REGION Network 16: Timeout
   Label( End_G7 )
   RUNG wire#powerrail
      Contact( #Switching_left )
      wire#w1
      { S7_Templates := "time_type := Time" } #MABS_sw_timout.TON(pt := T#10s, et =>)
      wire#w2
      I_Contact( #MABS.Reset_error )
      I_Contact( #MABS.EMS )
      Coil( #MABS.Error_timeout_sw )
   END_RUNG
   RUNG wire#powerrail
      Contact( #"Switching_left to straight" )
   END_RUNG wire#w1
   RUNG wire#powerrail
      Contact( #"Switching_right to straight" )
   END_RUNG wire#w1
   RUNG wire#powerrail
      Contact( #Switching_right )
   END_RUNG wire#w1
   RUNG wire#powerrail
      Contact( #MABS.Error_timeout_sw )
   END_RUNG wire#w2
   // the same network as SCL:
   End_G7:
   #MABS_sw_timout(IN := #Switching_left OR #"Switching_left to straight" OR #"Switching_right to straight" OR #Switching_right,   // TON
                   PT := T#10s);
   #MABS.Error_timeout_sw := (#MABS_sw_timout.Q OR #MABS.Error_timeout_sw) AND NOT #MABS.Reset_error AND NOT #MABS.EMS;
END_REGION

REGION Network 17: Postion reached + origin sensor
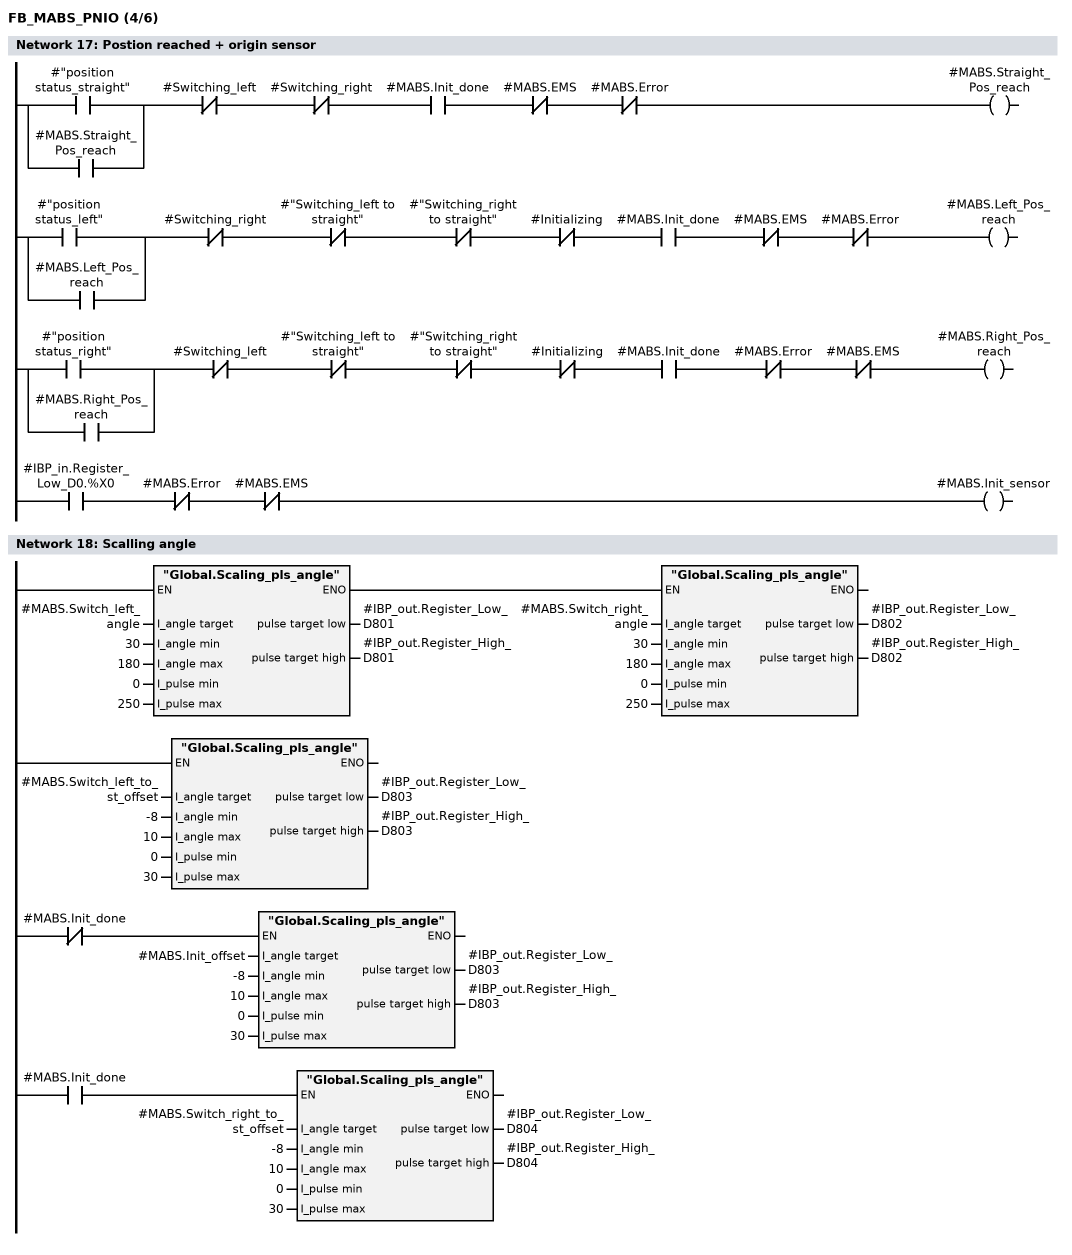
   RUNG wire#powerrail
      Contact( #"position status_straight" )
      wire#w1
      I_Contact( #Switching_left )
      I_Contact( #Switching_right )
      Contact( #MABS.Init_done )
      I_Contact( #MABS.EMS )
      I_Contact( #MABS.Error )
      Coil( #MABS.Straight_Pos_reach )
   END_RUNG
   RUNG wire#powerrail
      Contact( #MABS.Straight_Pos_reach )
   END_RUNG wire#w1
   RUNG wire#powerrail
      Contact( #"position status_left" )
      wire#w2
      I_Contact( #Switching_right )
      I_Contact( #"Switching_left to straight" )
      I_Contact( #"Switching_right to straight" )
      I_Contact( #Initializing )
      Contact( #MABS.Init_done )
      I_Contact( #MABS.EMS )
      I_Contact( #MABS.Error )
      Coil( #MABS.Left_Pos_reach )
   END_RUNG
   RUNG wire#powerrail
      Contact( #MABS.Left_Pos_reach )
   END_RUNG wire#w2
   RUNG wire#powerrail
      Contact( #"position status_right" )
      wire#w3
      I_Contact( #Switching_left )
      I_Contact( #"Switching_left to straight" )
      I_Contact( #"Switching_right to straight" )
      I_Contact( #Initializing )
      Contact( #MABS.Init_done )
      I_Contact( #MABS.Error )
      I_Contact( #MABS.EMS )
      Coil( #MABS.Right_Pos_reach )
   END_RUNG
   RUNG wire#powerrail
      Contact( #MABS.Right_Pos_reach )
   END_RUNG wire#w3
   RUNG wire#powerrail
      Contact( #IBP_in.Register_Low_D0.%X0 )
      I_Contact( #MABS.Error )
      I_Contact( #MABS.EMS )
      Coil( #MABS.Init_sensor )
   END_RUNG
   // the same network as SCL:
   #MABS.Straight_Pos_reach := (#"position status_straight" OR #MABS.Straight_Pos_reach) AND NOT #Switching_left AND NOT #Switching_right AND #MABS.Init_done AND NOT #MABS.EMS AND NOT #MABS.Error;
   #MABS.Left_Pos_reach := (#"position status_left" OR #MABS.Left_Pos_reach) AND NOT #Switching_right AND NOT #"Switching_left to straight" AND NOT #"Switching_right to straight" AND NOT #Initializing AND #MABS.Init_done AND NOT #MABS.EMS AND NOT #MABS.Error;
   #MABS.Right_Pos_reach := (#"position status_right" OR #MABS.Right_Pos_reach) AND NOT #Switching_left AND NOT #"Switching_left to straight" AND NOT #"Switching_right to straight" AND NOT #Initializing AND #MABS.Init_done AND NOT #MABS.Error AND NOT #MABS.EMS;
   #MABS.Init_sensor := #IBP_in.Register_Low_D0.%X0 AND NOT #MABS.Error AND NOT #MABS.EMS;
END_REGION

REGION Network 18: Scalling angle
   RUNG wire#powerrail
      "Global.Scaling_pls_angle"("I_angle target" := #MABS.Switch_left_angle, "I_angle min" := 30, "I_angle max" := 180, "I_pulse min" := 0, "I_pulse max" := 250, "pulse target low" => #IBP_out.Register_Low_D801, "pulse target high" => #IBP_out.Register_High_D801)
      "Global.Scaling_pls_angle"("I_angle target" := #MABS.Switch_right_angle, "I_angle min" := 30, "I_angle max" := 180, "I_pulse min" := 0, "I_pulse max" := 250, "pulse target low" => #IBP_out.Register_Low_D802, "pulse target high" => #IBP_out.Register_High_D802)
   END_RUNG
   RUNG wire#powerrail
      "Global.Scaling_pls_angle"("I_angle target" := #MABS.Switch_left_to_st_offset, "I_angle min" := -8, "I_angle max" := 10, "I_pulse min" := 0, "I_pulse max" := 30, "pulse target low" => #IBP_out.Register_Low_D803, "pulse target high" => #IBP_out.Register_High_D803)
   END_RUNG
   RUNG wire#powerrail
      I_Contact( #MABS.Init_done )
      "Global.Scaling_pls_angle"("I_angle target" := #MABS.Init_offset, "I_angle min" := -8, "I_angle max" := 10, "I_pulse min" := 0, "I_pulse max" := 30, "pulse target low" => #IBP_out.Register_Low_D803, "pulse target high" => #IBP_out.Register_High_D803)
   END_RUNG
   RUNG wire#powerrail
      Contact( #MABS.Init_done )
      "Global.Scaling_pls_angle"("I_angle target" := #MABS.Switch_right_to_st_offset, "I_angle min" := -8, "I_angle max" := 10, "I_pulse min" := 0, "I_pulse max" := 30, "pulse target low" => #IBP_out.Register_Low_D804, "pulse target high" => #IBP_out.Register_High_D804)
   END_RUNG
   // the same network as SCL:
   "Global.Scaling_pls_angle"("I_angle target" := #MABS.Switch_left_angle,
                           "I_angle min" := 30,
                           "I_angle max" := 180,
                           "I_pulse min" := 0,
                           "I_pulse max" := 250,
                           "pulse target low" => #IBP_out.Register_Low_D801,
                           "pulse target high" => #IBP_out.Register_High_D801,
                           ENO => #_w1);
   IF #_w1 THEN
       "Global.Scaling_pls_angle"("I_angle target" := #MABS.Switch_right_angle,
                               "I_angle min" := 30,
                               "I_angle max" := 180,
                               "I_pulse min" := 0,
                               "I_pulse max" := 250,
                               "pulse target low" => #IBP_out.Register_Low_D802,
                               "pulse target high" => #IBP_out.Register_High_D802);
   END_IF;
   "Global.Scaling_pls_angle"("I_angle target" := #MABS.Switch_left_to_st_offset,
                           "I_angle min" := -8,
                           "I_angle max" := 10,
                           "I_pulse min" := 0,
                           "I_pulse max" := 30,
                           "pulse target low" => #IBP_out.Register_Low_D803,
                           "pulse target high" => #IBP_out.Register_High_D803);
   IF NOT #MABS.Init_done THEN
       "Global.Scaling_pls_angle"("I_angle target" := #MABS.Init_offset,
                               "I_angle min" := -8,
                               "I_angle max" := 10,
                               "I_pulse min" := 0,
                               "I_pulse max" := 30,
                               "pulse target low" => #IBP_out.Register_Low_D803,
                               "pulse target high" => #IBP_out.Register_High_D803);
   END_IF;
   IF #MABS.Init_done THEN
       "Global.Scaling_pls_angle"("I_angle target" := #MABS.Switch_right_to_st_offset,
                               "I_angle min" := -8,
                               "I_angle max" := 10,
                               "I_pulse min" := 0,
                               "I_pulse max" := 30,
                               "pulse target low" => #IBP_out.Register_Low_D804,
                               "pulse target high" => #IBP_out.Register_High_D804);
   END_IF;
END_REGION

REGION Network 19: Swing direction
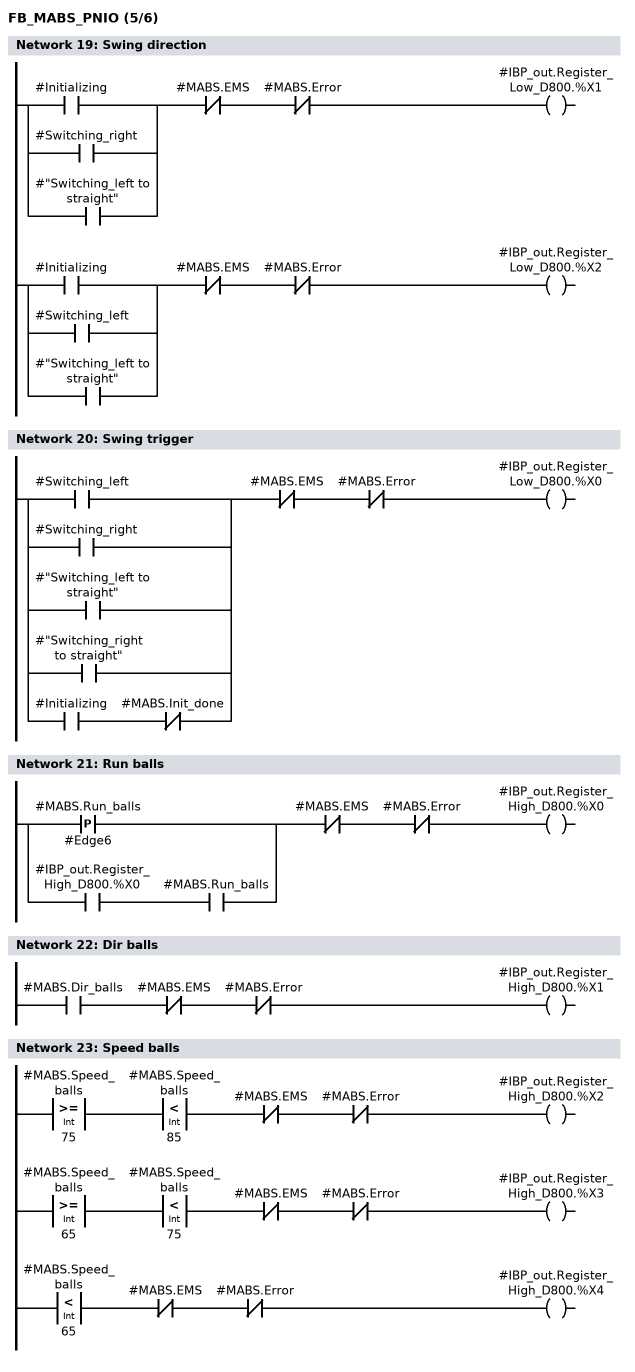
   RUNG wire#powerrail
      Contact( #Initializing )
      wire#w1
      I_Contact( #MABS.EMS )
      I_Contact( #MABS.Error )
      Coil( #IBP_out.Register_Low_D800.%X1 )
   END_RUNG
   RUNG wire#powerrail
      Contact( #Switching_right )
   END_RUNG wire#w1
   RUNG wire#powerrail
      Contact( #"Switching_left to straight" )
   END_RUNG wire#w1
   RUNG wire#powerrail
      Contact( #Initializing )
      wire#w2
      I_Contact( #MABS.EMS )
      I_Contact( #MABS.Error )
      Coil( #IBP_out.Register_Low_D800.%X2 )
   END_RUNG
   RUNG wire#powerrail
      Contact( #Switching_left )
   END_RUNG wire#w2
   RUNG wire#powerrail
      Contact( #"Switching_left to straight" )
   END_RUNG wire#w2
   // the same network as SCL:
   #IBP_out.Register_Low_D800.%X1 := (#Initializing OR #Switching_right OR #"Switching_left to straight") AND NOT #MABS.EMS AND NOT #MABS.Error;
   #IBP_out.Register_Low_D800.%X2 := (#Initializing OR #Switching_left OR #"Switching_left to straight") AND NOT #MABS.EMS AND NOT #MABS.Error;
END_REGION

REGION Network 20: Swing trigger
   RUNG wire#powerrail
      Contact( #Switching_left )
      wire#w1
      I_Contact( #MABS.EMS )
      I_Contact( #MABS.Error )
      Coil( #IBP_out.Register_Low_D800.%X0 )
   END_RUNG
   RUNG wire#powerrail
      Contact( #Switching_right )
   END_RUNG wire#w1
   RUNG wire#powerrail
      Contact( #"Switching_left to straight" )
   END_RUNG wire#w1
   RUNG wire#powerrail
      Contact( #"Switching_right to straight" )
   END_RUNG wire#w1
   RUNG wire#powerrail
      Contact( #Initializing )
      I_Contact( #MABS.Init_done )
   END_RUNG wire#w1
   // the same network as SCL:
   #IBP_out.Register_Low_D800.%X0 := (#Switching_left OR #Switching_right OR #"Switching_left to straight" OR #"Switching_right to straight" OR (#Initializing AND NOT #MABS.Init_done)) AND NOT #MABS.EMS AND NOT #MABS.Error;
END_REGION

REGION Network 21: Run balls
   RUNG wire#powerrail
      P_Contact(operand := #MABS.Run_balls, bit := #Edge6)
      wire#w1
      I_Contact( #MABS.EMS )
      I_Contact( #MABS.Error )
      Coil( #IBP_out.Register_High_D800.%X0 )
   END_RUNG
   RUNG wire#powerrail
      Contact( #IBP_out.Register_High_D800.%X0 )
      Contact( #MABS.Run_balls )
   END_RUNG wire#w1
   // the same network as SCL:
   #_w1 := #MABS.Run_balls AND NOT #Edge6;   // rising edge of #MABS.Run_balls
   #Edge6 := #MABS.Run_balls;
   #IBP_out.Register_High_D800.%X0 := (#_w1 OR (#IBP_out.Register_High_D800.%X0 AND #MABS.Run_balls)) AND NOT #MABS.EMS AND NOT #MABS.Error;
END_REGION

REGION Network 22: Dir balls
   RUNG wire#powerrail
      Contact( #MABS.Dir_balls )
      I_Contact( #MABS.EMS )
      I_Contact( #MABS.Error )
      Coil( #IBP_out.Register_High_D800.%X1 )
   END_RUNG
   // the same network as SCL:
   #IBP_out.Register_High_D800.%X1 := #MABS.Dir_balls AND NOT #MABS.EMS AND NOT #MABS.Error;
END_REGION

REGION Network 23: Speed balls
   RUNG wire#powerrail
      { S7_Templates := "SrcType := Int" } GE_Contact(in1 := #MABS.Speed_balls, in2 := 75)
      { S7_Templates := "SrcType := Int" } LT_Contact(in1 := #MABS.Speed_balls, in2 := 85)
      I_Contact( #MABS.EMS )
      I_Contact( #MABS.Error )
      Coil( #IBP_out.Register_High_D800.%X2 )
   END_RUNG
   RUNG wire#powerrail
      { S7_Templates := "SrcType := Int" } GE_Contact(in1 := #MABS.Speed_balls, in2 := 65)
      { S7_Templates := "SrcType := Int" } LT_Contact(in1 := #MABS.Speed_balls, in2 := 75)
      I_Contact( #MABS.EMS )
      I_Contact( #MABS.Error )
      Coil( #IBP_out.Register_High_D800.%X3 )
   END_RUNG
   RUNG wire#powerrail
      { S7_Templates := "SrcType := Int" } LT_Contact(in1 := #MABS.Speed_balls, in2 := 65)
      I_Contact( #MABS.EMS )
      I_Contact( #MABS.Error )
      Coil( #IBP_out.Register_High_D800.%X4 )
   END_RUNG
   // the same network as SCL:
   #IBP_out.Register_High_D800.%X2 := (#MABS.Speed_balls >= 75) AND (#MABS.Speed_balls < 85) AND NOT #MABS.EMS AND NOT #MABS.Error;
   #IBP_out.Register_High_D800.%X3 := (#MABS.Speed_balls >= 65) AND (#MABS.Speed_balls < 75) AND NOT #MABS.EMS AND NOT #MABS.Error;
   #IBP_out.Register_High_D800.%X4 := (#MABS.Speed_balls < 65) AND NOT #MABS.EMS AND NOT #MABS.Error;
END_REGION

REGION Network 24: HMI status
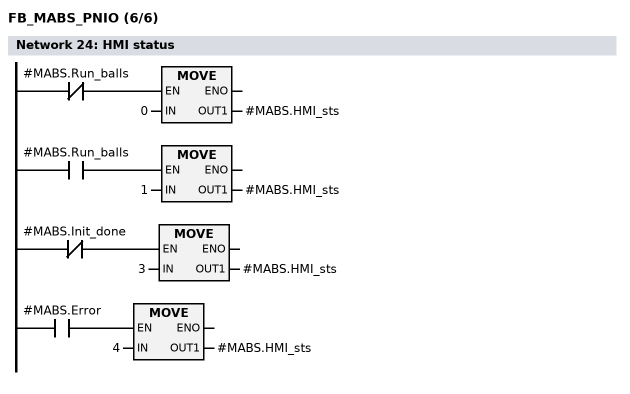
   RUNG wire#powerrail
      I_Contact( #MABS.Run_balls )
      Move(in := 0, out1 => #MABS.HMI_sts)
   END_RUNG
   RUNG wire#powerrail
      Contact( #MABS.Run_balls )
      Move(in := 1, out1 => #MABS.HMI_sts)
   END_RUNG
   RUNG wire#powerrail
      I_Contact( #MABS.Init_done )
      Move(in := 3, out1 => #MABS.HMI_sts)
   END_RUNG
   RUNG wire#powerrail
      Contact( #MABS.Error )
      Move(in := 4, out1 => #MABS.HMI_sts)
   END_RUNG
   // the same network as SCL:
   IF NOT #MABS.Run_balls THEN #MABS.HMI_sts := 0; END_IF;
   IF #MABS.Run_balls THEN #MABS.HMI_sts := 1; END_IF;
   IF NOT #MABS.Init_done THEN #MABS.HMI_sts := 3; END_IF;
   IF #MABS.Error THEN #MABS.HMI_sts := 4; END_IF;
END_REGION
END_FUNCTION_BLOCK

FUNCTION "Scaling_pls_angle" : Void   // FC12, LAD
// stored: Namespace Global, SetENOAutomatically false
   VAR_INPUT
      "I_angle target" : Int;
      "I_angle min" : Int;
      "I_angle max" : Int;
      "I_pulse min" : Int;
      "I_pulse max" : Int;
   END_VAR
   VAR_OUTPUT
      "pulse target low" : Byte;
      "pulse target high" : Byte;
   END_VAR
   VAR_TEMP
      R_pulse_calcul : Real;
      R_angle_calcul : Real;
      pulse_target_int : Int;
      Int4 : Int;
      Int5 : Int;
      Real1 : Real;
      Real2 : Real;
      Real3 : Real;
      Real4 : Real;
   END_VAR
BEGIN

REGION Network 1: Convert diff in real
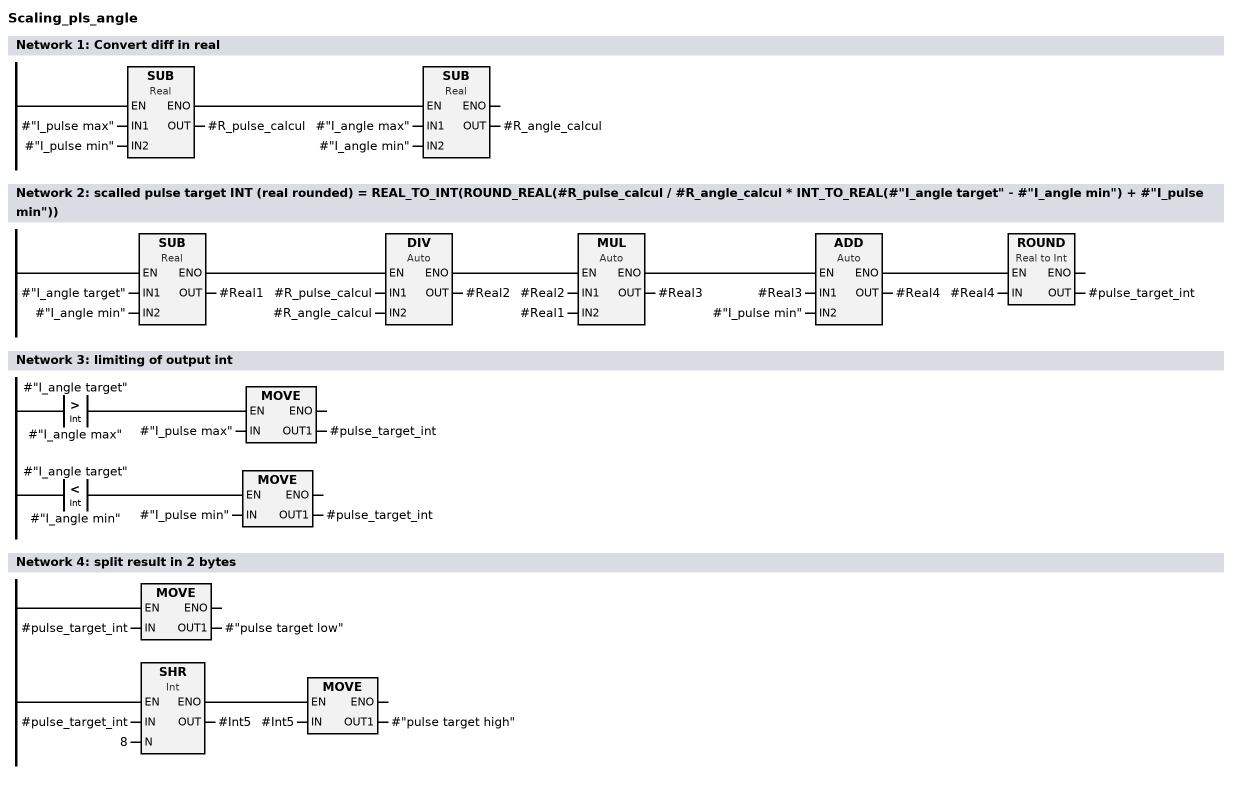
   RUNG wire#powerrail
      { S7_Templates := "SrcType := Real" } Sub(in1 := #"I_pulse max", in2 := #"I_pulse min", out => #R_pulse_calcul)
      { S7_Templates := "SrcType := Real" } Sub(in1 := #"I_angle max", in2 := #"I_angle min", out => #R_angle_calcul)
   END_RUNG
   // the same network as SCL:
   #R_pulse_calcul := #"I_pulse max" - #"I_pulse min";
   #R_angle_calcul := #"I_angle max" - #"I_angle min";
END_REGION

REGION Network 2: scalled pulse target INT (real rounded) = REAL_TO_INT(ROUND_REAL(#R_pulse_calcul / #R_angle_calcul * INT_TO_REAL(#"I_angle target" - #"I_angle min") + #"I_pulse min"))
   RUNG wire#powerrail
      { S7_Templates := "SrcType := Real" } Sub(in1 := #"I_angle target", in2 := #"I_angle min", out => #Real1)
      Div(in1 := #R_pulse_calcul, in2 := #R_angle_calcul, out => #Real2)
      Mul(in1 := #Real2, in2 := #Real1, out => #Real3)
      Add(in1 := #Real3, in2 := #"I_pulse min", out => #Real4)
      { S7_Templates := "[SrcType := Real, DestType := Int]" } Round(in := #Real4, out => #pulse_target_int)
   END_RUNG
   // the same network as SCL:
   #Real1 := #"I_angle target" - #"I_angle min";
   #Real2 := #R_pulse_calcul / #R_angle_calcul;
   #Real3 := #Real2 * #Real1;
   #Real4 := #Real3 + #"I_pulse min";
   #pulse_target_int := ROUND(#Real4);
END_REGION

REGION Network 3: limiting of output int
   RUNG wire#powerrail
      { S7_Templates := "SrcType := Int" } GT_Contact(in1 := #"I_angle target", in2 := #"I_angle max")
      Move(in := #"I_pulse max", out1 => #pulse_target_int)
   END_RUNG
   RUNG wire#powerrail
      { S7_Templates := "SrcType := Int" } LT_Contact(in1 := #"I_angle target", in2 := #"I_angle min")
      Move(in := #"I_pulse min", out1 => #pulse_target_int)
   END_RUNG
   // the same network as SCL:
   IF #"I_angle target" > #"I_angle max" THEN #pulse_target_int := #"I_pulse max"; END_IF;
   IF #"I_angle target" < #"I_angle min" THEN #pulse_target_int := #"I_pulse min"; END_IF;
END_REGION

REGION Network 4: split result in 2 bytes
   RUNG wire#powerrail
      Move(in := #pulse_target_int, out1 => #"pulse target low")
   END_RUNG
   RUNG wire#powerrail
      { S7_Templates := "SrcType := Int" } Shr(in := #pulse_target_int, n := 8, out => #Int5)
      Move(in := #Int5, out1 => #"pulse target high")
   END_RUNG
   // the same network as SCL:
   #"pulse target low" := #pulse_target_int;
   #Int5 := SHR(IN := #pulse_target_int, N := 8);
   #"pulse target high" := #Int5;
END_REGION
END_FUNCTION

FUNCTION_BLOCK "FB_ManualControl"   // FB37, LAD
// stored: Access Published, MemoryReserve 100, Namespace Global, SetENOAutomatically false
   VAR RETAIN
      "Counter" { S7_SetPoint := 'True'} : CTU_INT;
   END_VAR
BEGIN

REGION Network 1
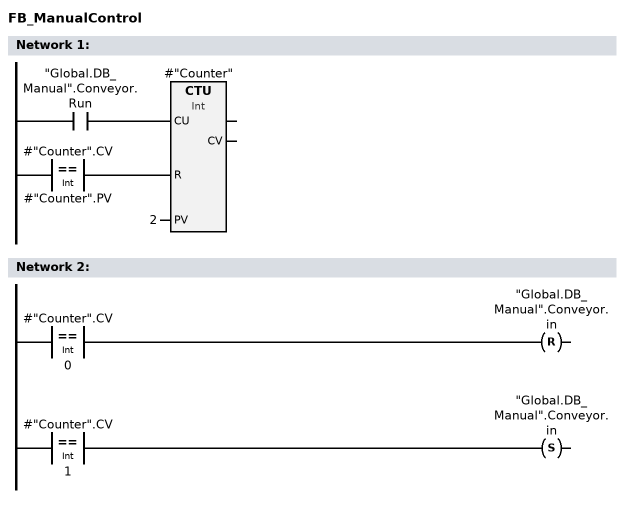
   RUNG wire#powerrail
      Contact( "Global.DB_Manual".Conveyor.Run )
      { S7_Templates := "value_type := Int" } #"Counter".CTU(r := wire#w1, pv := 2, cv =>)
   END_RUNG
   RUNG wire#powerrail
      { S7_Templates := "SrcType := Int" } EQ_Contact(in1 := #"Counter".CV, in2 := #"Counter".PV)
   END_RUNG wire#w1
   // the same network as SCL:
   #"Counter"(CU := "Global.DB_Manual".Conveyor.Run, R := #"Counter".CV = #"Counter".PV, PV := 2);   // CTU
END_REGION

REGION Network 2
   RUNG wire#powerrail
      { S7_Templates := "SrcType := Int" } EQ_Contact(in1 := #"Counter".CV, in2 := 0)
      R_Coil( "Global.DB_Manual".Conveyor.in )
   END_RUNG
   RUNG wire#powerrail
      { S7_Templates := "SrcType := Int" } EQ_Contact(in1 := #"Counter".CV, in2 := 1)
      S_Coil( "Global.DB_Manual".Conveyor.in )
   END_RUNG
   // the same network as SCL:
   IF #"Counter".CV = 0 THEN "Global.DB_Manual".Conveyor.in := FALSE; END_IF;
   IF #"Counter".CV = 1 THEN "Global.DB_Manual".Conveyor.in := TRUE; END_IF;
END_REGION
END_FUNCTION_BLOCK

FUNCTION "FC_SafetyStandard" : Void
{ S7_Optimized_Access := 'TRUE' ; Published := 'TRUE' }
VERSION : 0.1

BEGIN
END_FUNCTION

NAMESPACE Global
ORGANIZATION_BLOCK Main_OB
TITLE = "Main Program Sweep (Cycle)"
{ S7_Optimized_Access := 'TRUE' ; Published := 'FALSE' }
VERSION : 0.1

BEGIN
	// ===
	// GoW
	// ==========================================================================================================================================
	// Company        : LogTech, s.r.o.
	// Created by     : Anton Vinoth Soundraraj
	// Block          : Main_OB
	// Project        : Lékarna DC Chrudim
	// Project number : 23-157
	// ==========================================================================================================================================
	
	REGION System
	    
	    FC_ReadSystemSSR();
	    
	END_REGION
	
	REGION Hardware diag
	    
	    IDB_HardwareDiag();
	    
	END_REGION
	
	REGION Klaxon
	    
	    FC_AllKlaxon();
	    
	END_REGION
	
	REGION Devices
	    
	    IDB_DataMan262(TriggerSignal:=DB_SystemSimu.TriggerSensor.Line.C1.Conveyor[3001],
	                   "Dataman-Results Available":=_."Dataman-Results Available",
	                   "Dataman-TriggerReady":=_."Dataman-TriggerReady",
	                   "Dataman-TriggerAck":=_."Dataman-TriggerAck",
	                   "Dataman-ResultID":=_."Dataman-ResultID",
	                   "Dataman-Result Code":=_."Dataman-Result Code",
	                   "Dataman-Result Length":=_."Dataman-Result Length",
	                   "Result Data":=_."Result Data",
	                   "Dataman-UserData Length"=>_."Dataman-UserData Length",
	                   "Dataman-UserData Option"=>_."Dataman-UserData Option",
	                   "User Data"=>_."User Data",
	                   "Dataman-TriggerEnable":=_."Dataman-TriggerEnable",
	                   "Dataman-Trigger":=_."Dataman-Trigger",
	                   "Dataman-ResultsAck":=_."Dataman-ResultsAck");
	    
	END_REGION
	
END_ORGANIZATION_BLOCK
END_NAMESPACE

NAMESPACE LineA1
FUNCTION_BLOCK FB_LineA1
{ S7_Optimized_Access := 'TRUE' ; Published := 'TRUE' }
VERSION : 0.1
   VAR 
      "Conveyor_A1.1.1" { S7_SetPoint := 'False'} : _.Global.FB_Conveyor;
      "MABS_A1.1.1" { S7_SetPoint := 'False'} : _.Global.FB_MABS;
      "Transfer_A1.1.1" { S7_SetPoint := 'False'} : _.Global.FB_S300_tTransMode;
   END_VAR


BEGIN
	
	
	
	
	
	
	
	
	
	
	
	
	
	
	
END_FUNCTION_BLOCK
END_NAMESPACE

NAMESPACE LineA1
ORGANIZATION_BLOCK Main_LineA1
TITLE = "Main Program Sweep (Cycle)"
{ S7_Optimized_Access := 'TRUE' ; Published := 'FALSE' }
VERSION : 0.1

BEGIN
	IDB_LineA1();
	
END_ORGANIZATION_BLOCK
END_NAMESPACE

NAMESPACE LineB1
FUNCTION_BLOCK FB_LineB1
{ S7_Optimized_Access := 'TRUE' ; Published := 'TRUE' }
VERSION : 0.1
   VAR 
      "Conveyor_B1.1.1" { S7_SetPoint := 'False'} : _.Global.FB_Conveyor;
      "MABS_B1.1.1" { S7_SetPoint := 'False'} : _.Global.FB_MABS;
      "Transfer_B1.1.1" { S7_SetPoint := 'False'} : _.Global.FB_S300_tTransMode;
      "Transfer_B1.1.2" { S7_SetPoint := 'False'} : FB_S300_FullControl;
   END_VAR


BEGIN
	
	
	
	
	
	
	
	
	
	
	
	
	
	
	
END_FUNCTION_BLOCK
END_NAMESPACE

NAMESPACE LineB1
ORGANIZATION_BLOCK Main_LineB1
TITLE = "Main Program Sweep (Cycle)"
{ S7_Optimized_Access := 'TRUE' ; Published := 'FALSE' }
VERSION : 0.1

BEGIN
	IDB_LineB1();
	
END_ORGANIZATION_BLOCK
END_NAMESPACE

NAMESPACE LineC1
FUNCTION_BLOCK FB_LineC1
{ S7_Optimized_Access := 'TRUE' ; Published := 'TRUE' }
VERSION : 0.1
   VAR 
      "Conveyor_C1.1.1" { S7_SetPoint := 'False'} : _.Global.FB_Conveyor;
      "Conveyor_C1.1.2" : _.Global.FB_Conveyor;
      "Conveyor_C1.1.3" : _.Global.FB_Conveyor;
      "MABS_C1.2.1" { S7_SetPoint := 'False'} : _.Global.FB_MABS;
      "MABS_C1.2.2" : _.Global.FB_MABS;
      "Conveyor_C1.3.1" : _.Global.FB_Conveyor;
      "Conveyor_C1.3.2" : _.Global.FB_Conveyor;
      "Conveyor_C1.3.3" : _.Global.FB_Conveyor;
      "Conveyor_C1.3.4" : _.Global.FB_Conveyor;
      "Conveyor_C1.3.5" : _.Global.FB_Conveyor;
      "Conveyor_C1.3.6" : _.Global.FB_Conveyor;
      "Conveyor_C1.3.7" : _.Global.FB_Conveyor;
      "Conveyor_C1.3.8" : _.Global.FB_Conveyor;
      "Conveyor_C1.3.9" : _.Global.FB_Conveyor;
      "Conveyor_C1.3.10" : _.Global.FB_Conveyor;
      "Conveyor_C1.4.1" : _.Global.FB_Conveyor;
      "Conveyor_C1.4.2" : _.Global.FB_Conveyor;
      "Conveyor_C1.4.3" : _.Global.FB_Conveyor;
      "Conveyor_C1.4.4" : _.Global.FB_Conveyor;
      "Conveyor_C1.5.1" : _.Global.FB_Conveyor;
      "Conveyor_C1.6.1" : _.Global.FB_Conveyor;
      "Conveyor_C1.6.2" : _.Global.FB_Conveyor;
      "Conveyor_C1.7.1" : _.Global.FB_Conveyor;
      "Conveyor_C1.7.2" : _.Global.FB_Conveyor;
      "Conveyor_C1.7.3" : _.Global.FB_Conveyor;
      "Conveyor_C1.7.4" : _.Global.FB_Conveyor;
      "Conveyor_C1.7.5" : _.Global.FB_Conveyor;
      "Conveyor_C1.7.6" : _.Global.FB_Conveyor;
      "Conveyor_C1.7.7" : _.Global.FB_Conveyor;
      "Conveyor_C1.7.8" : _.Global.FB_Conveyor;
      "Conveyor_C1.7.9" : _.Global.FB_Conveyor;
      "Conveyor_C1.7.10" : _.Global.FB_Conveyor;
      "Conveyor_C1.8.0" : _.Global.FB_Conveyor;
      "Conveyor_C1.9.1" : _.Global.FB_Conveyor;
      "Conveyor_C1.10.1" : _.Global.FB_Conveyor;
      "Conveyor_C1.11.1" : _.Global.FB_Conveyor;
      "Conveyor_C1.11.2" : _.Global.FB_Conveyor;
      "Conveyor_C1.12.1" : _.Global.FB_Conveyor;
      "Conveyor_C1.12.2" : _.Global.FB_Conveyor;
      "Conveyor_C1.12.3" : _.Global.FB_Conveyor;
      "Transfer_C1.13.1" { S7_SetPoint := 'False'} : _.Global.FB_S300_tTransMode;
      "Transfer_C1.14.1" : _.Global.FB_S300_tTransMode;
      "Conveyor_C1.15.2" : _.Global.FB_Conveyor;
      "Conveyor_C1.15.3" : _.Global.FB_Conveyor;
      "Conveyor_C1.15.4" : _.Global.FB_Conveyor;
      "Conveyor_C1.16.1" : _.Global.FB_Conveyor;
      "Conveyor_C1.17.0" : _.Global.FB_Conveyor;
      "Conveyor_C1.18.1" : _.Global.FB_Conveyor;
      "Conveyor_C1.18.2" : _.Global.FB_Conveyor;
      "Conveyor_C1.18.3" : _.Global.FB_Conveyor;
      "Conveyor_C1.18.4" : _.Global.FB_Conveyor;
      "Conveyor_C1.18.5" : _.Global.FB_Conveyor;
      "Conveyor_C1.18.6" : _.Global.FB_Conveyor;
      "Conveyor_C1.18.7" : _.Global.FB_Conveyor;
      "Conveyor_C1.19.1" : _.Global.FB_Conveyor;
      "Conveyor_C1.20.2" : _.Global.FB_Conveyor;
   END_VAR


BEGIN
	// ==========================================================================================================================================
	// Company        : LogTech, s.r.o.
	// Created by     : Mahmoud Elnady
	// Block          : FC_UpstreaProductionTote
	// Project        : Lekarna, Chrudim -PLC001 -MCC001
	// Project number : 23-157
	// ==========================================================================================================================================
	//start this comment 
	REGION Conveyor_C1.1.1
	    #"Conveyor_C1.1.1"(ConveyorID := _."Conveyor_C1.1.1",
	                       Fault := _.LineC1.DB_UDI.LineC1.Fault.Conveyor[_."Conveyor_C1.1.1"],
	                       Upstream := _.LineC1.DB_UDI.LineC1.Upstream.Conveyor[_."Conveyor_C1.1.1"],
	                       Downstream := _.LineC1.DB_UDI.LineC1.DownstreamAccu.Conveyor[_."Conveyor_C1.1.1"],
	                       Interlock := _.LineC1.DB_UDI.LineC1.Interlock.Conveyor[_."Conveyor_C1.1.1"]);
	END_REGION
	
	
	
	
	REGION Conveyor_C1.1.2
	    #"Conveyor_C1.1.2"(ConveyorID := _."Conveyor_C1.1.2",
	                       Fault := _.LineC1.DB_UDI.LineC1.Fault.Conveyor[_."Conveyor_C1.1.2"],
	                       Upstream := _.LineC1.DB_UDI.LineC1.Upstream.Conveyor[_."Conveyor_C1.1.2"],
	                       Downstream := _.LineC1.DB_UDI.LineC1.DownstreamAccu.Conveyor[_."Conveyor_C1.1.2"],
	                       Interlock := _.LineC1.DB_UDI.LineC1.Interlock.Conveyor[_."Conveyor_C1.1.2"]);
	    ;
	END_REGION
	
	
	
	REGION Conveyor_C1.1.3
	    #"Conveyor_C1.1.3"(ConveyorID := _."Conveyor_C1.1.3",
	                       Fault := _.LineC1.DB_UDI.LineC1.Fault.Conveyor[_."Conveyor_C1.1.3"],
	                       Upstream := _.LineC1.DB_UDI.LineC1.Upstream.Conveyor[_."Conveyor_C1.1.3"],
	                       Downstream := _.LineC1.DB_UDI.LineC1.DownstreamAccu.Conveyor[_."Conveyor_C1.1.3"],
	                       Interlock := _.LineC1.DB_UDI.LineC1.Interlock.Conveyor[_."Conveyor_C1.1.3"]);
	    ;
	END_REGION
	
	
	
	REGION MABS_C1.2.1
	    #"MABS_C1.2.1"(MABS_ID:=_."MABS_C1.2.1",
	                   CrossSensor:=false,
	                   Fault:=_.LineC1.DB_UDI.LineC1.Fault.Conveyor[_."MABS_C1.2.1"],
	                   UpstreamRunning:= #"Conveyor_C1.1.3".ReadConveyorStatus.Running,
	                   Downstream_Straight:=#"Conveyor_C1.3.1".FilteredSensor,
	                   "Downstream_Right/Left":=#"Conveyor_C1.9.1".FilteredSensor,
	                   SortDir:= _.Global.DB_ToteTracking.Conveyor[_."MABS_C1.2.1"].ToteDir,
	                   Setpoints:=DB_ConveyorParameters.Line.C1.MABS[_."MABS_C1.2.1"],
	                   MABS_IBP_in:=_."MABS_C1.2.1_IN",
	                   MABS_IBP_out:=_."MABS_C1.2.1_Out");
	END_REGION
	
	
	
	REGION MABS_C1.2.2
	    #"MABS_C1.2.2"(MABS_ID := _."MABS_C1.2.2",
	                   CrossSensor := false,
	                   Fault := _.LineC1.DB_UDI.LineC1.Fault.Conveyor[_."MABS_C1.2.2"],
	                   UpstreamRunning := #"Conveyor_C1.1.3".ReadConveyorStatus.Running,
	                   Downstream_Straight := #"Conveyor_C1.3.1".FilteredSensor,
	                   "Downstream_Right/Left" := #"Conveyor_C1.9.1".FilteredSensor,
	                   SortDir := _.Global.DB_ToteTracking.Conveyor[_."MABS_C1.2.2"].ToteDir,
	                   Setpoints := DB_ConveyorParameters.Line.C1.MABS[_."MABS_C1.2.2"],
	                   MABS_IBP_in := _."MABS_C1.2.2_IN",
	                   MABS_IBP_out := _."MABS_C1.2.2_Out");
	END_REGION
	
	
	REGION Conveyor_C1.3.1
	    #"Conveyor_C1.3.1"(ConveyorID := _."Conveyor_C1.3.1",
	                       Fault := _.LineC1.DB_UDI.LineC1.Fault.Conveyor[_."Conveyor_C1.3.1"],
	                       Upstream := _.LineC1.DB_UDI.LineC1.Upstream.Conveyor[_."Conveyor_C1.3.1"],
	                       Downstream := _.LineC1.DB_UDI.LineC1.DownstreamAccu.Conveyor[_."Conveyor_C1.3.1"],
	                       Interlock := _.LineC1.DB_UDI.LineC1.Interlock.Conveyor[_."Conveyor_C1.3.1"]);
	    ;
	END_REGION
	
	
	REGION Conveyor_C1.3.2
	    #"Conveyor_C1.3.2"(ConveyorID := _."Conveyor_C1.3.2",
	                       Fault := _.LineC1.DB_UDI.LineC1.Fault.Conveyor[_."Conveyor_C1.3.2"],
	                       Upstream := _.LineC1.DB_UDI.LineC1.Upstream.Conveyor[_."Conveyor_C1.3.2"],
	                       Downstream := _.LineC1.DB_UDI.LineC1.DownstreamAccu.Conveyor[_."Conveyor_C1.3.2"],
	                       Interlock := _.LineC1.DB_UDI.LineC1.Interlock.Conveyor[_."Conveyor_C1.3.2"]);
	    ;
	END_REGION
	
	
	REGION Conveyor_C1.3.3
	    #"Conveyor_C1.3.3"(ConveyorID := _."Conveyor_C1.3.3",
	                       Fault := _.LineC1.DB_UDI.LineC1.Fault.Conveyor[_."Conveyor_C1.3.3"],
	                       Upstream := _.LineC1.DB_UDI.LineC1.Upstream.Conveyor[_."Conveyor_C1.3.3"],
	                       Downstream := _.LineC1.DB_UDI.LineC1.DownstreamAccu.Conveyor[_."Conveyor_C1.3.3"],
	                       Interlock := _.LineC1.DB_UDI.LineC1.Interlock.Conveyor[_."Conveyor_C1.3.3"]);
	    ;
	END_REGION
	
	
	REGION Conveyor_C1.3.4
	    #"Conveyor_C1.3.4"(ConveyorID := _."Conveyor_C1.3.4",
	                       Fault := _.LineC1.DB_UDI.LineC1.Fault.Conveyor[_."Conveyor_C1.3.4"],
	                       Upstream := _.LineC1.DB_UDI.LineC1.Upstream.Conveyor[_."Conveyor_C1.3.4"],
	                       Downstream := _.LineC1.DB_UDI.LineC1.DownstreamAccu.Conveyor[_."Conveyor_C1.3.4"],
	                       Interlock := _.LineC1.DB_UDI.LineC1.Interlock.Conveyor[_."Conveyor_C1.3.4"]);
	    
	END_REGION
	
	
	REGION Conveyor_C1.3.5
	    #"Conveyor_C1.3.5"(ConveyorID := _."Conveyor_C1.3.5",
	                       Fault := _.LineC1.DB_UDI.LineC1.Fault.Conveyor[_."Conveyor_C1.3.5"],
	                       Upstream := _.LineC1.DB_UDI.LineC1.Upstream.Conveyor[_."Conveyor_C1.3.5"],
	                       Downstream := _.LineC1.DB_UDI.LineC1.DownstreamAccu.Conveyor[_."Conveyor_C1.3.5"],
	                       Interlock := _.LineC1.DB_UDI.LineC1.Interlock.Conveyor[_."Conveyor_C1.3.5"]);
	    ;
	END_REGION
	
	
	REGION Conveyor_C1.3.6
	    #"Conveyor_C1.3.6"(ConveyorID := _."Conveyor_C1.3.6",
	                       Fault := _.LineC1.DB_UDI.LineC1.Fault.Conveyor[_."Conveyor_C1.3.6"],
	                       Upstream := _.LineC1.DB_UDI.LineC1.Upstream.Conveyor[_."Conveyor_C1.3.6"],
	                       Downstream := _.LineC1.DB_UDI.LineC1.DownstreamAccu.Conveyor[_."Conveyor_C1.3.6"],
	                       Interlock := _.LineC1.DB_UDI.LineC1.Interlock.Conveyor[_."Conveyor_C1.3.6"]);
	    ;
	END_REGION
	
	
	REGION Conveyor_C1.3.7
	    #"Conveyor_C1.3.7"(ConveyorID := _."Conveyor_C1.3.7",
	                       Fault := _.LineC1.DB_UDI.LineC1.Fault.Conveyor[_."Conveyor_C1.3.7"],
	                       Upstream := _.LineC1.DB_UDI.LineC1.Upstream.Conveyor[_."Conveyor_C1.3.7"],
	                       Downstream := _.LineC1.DB_UDI.LineC1.DownstreamAccu.Conveyor[_."Conveyor_C1.3.7"],
	                       Interlock := _.LineC1.DB_UDI.LineC1.Interlock.Conveyor[_."Conveyor_C1.3.7"]);
	    ;
	END_REGION
	
	
	
	REGION Conveyor_C1.3.8
	    #"Conveyor_C1.3.8"(ConveyorID := _."Conveyor_C1.3.8",
	                       Fault := _.LineC1.DB_UDI.LineC1.Fault.Conveyor[_."Conveyor_C1.3.8"],
	                       Upstream := _.LineC1.DB_UDI.LineC1.Upstream.Conveyor[_."Conveyor_C1.3.8"],
	                       Downstream := _.LineC1.DB_UDI.LineC1.DownstreamAccu.Conveyor[_."Conveyor_C1.3.8"],
	                       Interlock := _.LineC1.DB_UDI.LineC1.Interlock.Conveyor[_."Conveyor_C1.3.8"]);
	    ;
	END_REGION
	
	
	REGION Conveyor_C1.3.9
	    #"Conveyor_C1.3.9"(ConveyorID := _."Conveyor_C1.3.9",
	                       Fault := _.LineC1.DB_UDI.LineC1.Fault.Conveyor[_."Conveyor_C1.3.9"],
	                       Upstream := _.LineC1.DB_UDI.LineC1.Upstream.Conveyor[_."Conveyor_C1.3.9"],
	                       Downstream := _.LineC1.DB_UDI.LineC1.DownstreamAccu.Conveyor[_."Conveyor_C1.3.9"],
	                       Interlock := _.LineC1.DB_UDI.LineC1.Interlock.Conveyor[_."Conveyor_C1.3.9"]);
	    ;
	END_REGION
	
	
	REGION Conveyor_C1.3.10
	    #"Conveyor_C1.3.10"(ConveyorID := _."Conveyor_C1.3.10",
	                        Fault := _.LineC1.DB_UDI.LineC1.Fault.Conveyor[_."Conveyor_C1.3.10"],
	                        Upstream := _.LineC1.DB_UDI.LineC1.Upstream.Conveyor[_."Conveyor_C1.3.10"],
	                        Downstream := _.LineC1.DB_UDI.LineC1.DownstreamAccu.Conveyor[_."Conveyor_C1.3.10"],
	                        Interlock := _.LineC1.DB_UDI.LineC1.Interlock.Conveyor[_."Conveyor_C1.3.10"]);
	    ;
	END_REGION
	
	
	REGION Conveyor_C1.4.1
	    #"Conveyor_C1.4.1"(ConveyorID := _."Conveyor_C1.4.1",
	                       Fault := _.LineC1.DB_UDI.LineC1.Fault.Conveyor[_."Conveyor_C1.4.1"],
	                       Upstream := _.LineC1.DB_UDI.LineC1.Upstream.Conveyor[_."Conveyor_C1.4.1"],
	                       Downstream := _.LineC1.DB_UDI.LineC1.DownstreamAccu.Conveyor[_."Conveyor_C1.4.1"],
	                       Interlock := _.LineC1.DB_UDI.LineC1.Interlock.Conveyor[_."Conveyor_C1.4.1"]);
	    ;
	END_REGION
	
	
	REGION Conveyor_C1.4.2
	    #"Conveyor_C1.4.2"(ConveyorID := _."Conveyor_C1.4.2",
	                       Fault := _.LineC1.DB_UDI.LineC1.Fault.Conveyor[_."Conveyor_C1.4.2"],
	                       Upstream := _.LineC1.DB_UDI.LineC1.Upstream.Conveyor[_."Conveyor_C1.4.2"],
	                       Downstream := _.LineC1.DB_UDI.LineC1.DownstreamAccu.Conveyor[_."Conveyor_C1.4.2"],
	                       Interlock := _.LineC1.DB_UDI.LineC1.Interlock.Conveyor[_."Conveyor_C1.4.2"]);
	    ;
	END_REGION
	
	
	REGION Conveyor_C1.4.3
	    #"Conveyor_C1.4.3"(ConveyorID := _."Conveyor_C1.4.3",
	                       Fault := _.LineC1.DB_UDI.LineC1.Fault.Conveyor[_."Conveyor_C1.4.3"],
	                       Upstream := _.LineC1.DB_UDI.LineC1.Upstream.Conveyor[_."Conveyor_C1.4.3"],
	                       Downstream := _.LineC1.DB_UDI.LineC1.DownstreamAccu.Conveyor[_."Conveyor_C1.4.3"],
	                       Interlock := _.LineC1.DB_UDI.LineC1.Interlock.Conveyor[_."Conveyor_C1.4.3"]);
	    ;
	END_REGION
	
	
	REGION Conveyor_C1.4.4
	    #"Conveyor_C1.4.4"(ConveyorID := _."Conveyor_C1.4.4",
	                       Fault := _.LineC1.DB_UDI.LineC1.Fault.Conveyor[_."Conveyor_C1.4.4"],
	                       Upstream := _.LineC1.DB_UDI.LineC1.Upstream.Conveyor[_."Conveyor_C1.4.4"],
	                       Downstream := _.LineC1.DB_UDI.LineC1.DownstreamAccu.Conveyor[_."Conveyor_C1.4.4"],
	                       Interlock := _.LineC1.DB_UDI.LineC1.Interlock.Conveyor[_."Conveyor_C1.4.4"]);
	    ;
	END_REGION
	
	
	REGION Conveyor_C1.5.1
	    #"Conveyor_C1.5.1"(ConveyorID := _."Conveyor_C1.5.1",
	                       Fault := _.LineC1.DB_UDI.LineC1.Fault.Conveyor[_."Conveyor_C1.5.1"],
	                       Upstream := _.LineC1.DB_UDI.LineC1.Upstream.Conveyor[_."Conveyor_C1.5.1"],
	                       Downstream := _.LineC1.DB_UDI.LineC1.DownstreamAccu.Conveyor[_."Conveyor_C1.5.1"],
	                       Interlock := _.LineC1.DB_UDI.LineC1.Interlock.Conveyor[_."Conveyor_C1.5.1"]);
	    ;
	END_REGION
	
	
	REGION Conveyor_C1.6.1
	    #"Conveyor_C1.6.1"(ConveyorID := _."Conveyor_C1.6.1",
	                       Fault := _.LineC1.DB_UDI.LineC1.Fault.Conveyor[_."Conveyor_C1.6.1"],
	                       Upstream := _.LineC1.DB_UDI.LineC1.Upstream.Conveyor[_."Conveyor_C1.6.1"],
	                       Downstream := _.LineC1.DB_UDI.LineC1.DownstreamAccu.Conveyor[_."Conveyor_C1.6.1"],
	                       Interlock := _.LineC1.DB_UDI.LineC1.Interlock.Conveyor[_."Conveyor_C1.6.1"]);
	    ;
	END_REGION
	
	
	REGION Conveyor_C1.6.2
	    #"Conveyor_C1.6.2"(ConveyorID := _."Conveyor_C1.6.2",
	                       Fault := _.LineC1.DB_UDI.LineC1.Fault.Conveyor[_."Conveyor_C1.6.2"],
	                       Upstream := _.LineC1.DB_UDI.LineC1.Upstream.Conveyor[_."Conveyor_C1.6.2"],
	                       Downstream := _.LineC1.DB_UDI.LineC1.DownstreamAccu.Conveyor[_."Conveyor_C1.6.2"],
	                       Interlock := _.LineC1.DB_UDI.LineC1.Interlock.Conveyor[_."Conveyor_C1.6.2"]);
	    ;
	END_REGION
	
	
	REGION Conveyor_C1.7.1
	    #"Conveyor_C1.7.1"(ConveyorID := _."Conveyor_C1.7.1",
	                       Fault := _.LineC1.DB_UDI.LineC1.Fault.Conveyor[_."Conveyor_C1.7.1"],
	                       Upstream := _.LineC1.DB_UDI.LineC1.Upstream.Conveyor[_."Conveyor_C1.7.1"],
	                       Downstream := _.LineC1.DB_UDI.LineC1.DownstreamAccu.Conveyor[_."Conveyor_C1.7.1"],
	                       Interlock := _.LineC1.DB_UDI.LineC1.Interlock.Conveyor[_."Conveyor_C1.7.1"]);
	    ;
	END_REGION
	
	
	REGION Conveyor_C1.7.2
	    #"Conveyor_C1.7.2"(ConveyorID := _."Conveyor_C1.7.2",
	                       Fault := _.LineC1.DB_UDI.LineC1.Fault.Conveyor[_."Conveyor_C1.7.2"],
	                       Upstream := _.LineC1.DB_UDI.LineC1.Upstream.Conveyor[_."Conveyor_C1.7.2"],
	                       Downstream := _.LineC1.DB_UDI.LineC1.DownstreamAccu.Conveyor[_."Conveyor_C1.7.2"],
	                       Interlock := _.LineC1.DB_UDI.LineC1.Interlock.Conveyor[_."Conveyor_C1.7.2"]);
	    ;
	END_REGION
	
	
	REGION Conveyor_C1.7.3
	    #"Conveyor_C1.7.3"(ConveyorID := _."Conveyor_C1.7.3",
	                       Fault := _.LineC1.DB_UDI.LineC1.Fault.Conveyor[_."Conveyor_C1.7.3"],
	                       Upstream := _.LineC1.DB_UDI.LineC1.Upstream.Conveyor[_."Conveyor_C1.7.3"],
	                       Downstream := _.LineC1.DB_UDI.LineC1.DownstreamAccu.Conveyor[_."Conveyor_C1.7.3"],
	                       Interlock := _.LineC1.DB_UDI.LineC1.Interlock.Conveyor[_."Conveyor_C1.7.3"]);
	    ;
	END_REGION
	
	
	REGION Conveyor_C1.7.4
	    #"Conveyor_C1.7.4"(ConveyorID := _."Conveyor_C1.7.4",
	                       Fault := _.LineC1.DB_UDI.LineC1.Fault.Conveyor[_."Conveyor_C1.7.4"],
	                       Upstream := _.LineC1.DB_UDI.LineC1.Upstream.Conveyor[_."Conveyor_C1.7.4"],
	                       Downstream := _.LineC1.DB_UDI.LineC1.DownstreamAccu.Conveyor[_."Conveyor_C1.7.4"],
	                       Interlock := _.LineC1.DB_UDI.LineC1.Interlock.Conveyor[_."Conveyor_C1.7.4"]);
	    ;
	END_REGION
	
	
	REGION Conveyor_C1.7.5
	    #"Conveyor_C1.7.5"(ConveyorID := _."Conveyor_C1.7.5",
	                       Fault := _.LineC1.DB_UDI.LineC1.Fault.Conveyor[_."Conveyor_C1.7.5"],
	                       Upstream := _.LineC1.DB_UDI.LineC1.Upstream.Conveyor[_."Conveyor_C1.7.5"],
	                       Downstream := _.LineC1.DB_UDI.LineC1.DownstreamAccu.Conveyor[_."Conveyor_C1.7.5"],
	                       Interlock := _.LineC1.DB_UDI.LineC1.Interlock.Conveyor[_."Conveyor_C1.7.5"]);
	    ;
	END_REGION
	
	
	REGION Conveyor_C1.7.6
	    #"Conveyor_C1.7.6"(ConveyorID := _."Conveyor_C1.7.6",
	                       Fault := _.LineC1.DB_UDI.LineC1.Fault.Conveyor[_."Conveyor_C1.7.6"],
	                       Upstream := _.LineC1.DB_UDI.LineC1.Upstream.Conveyor[_."Conveyor_C1.7.6"],
	                       Downstream := _.LineC1.DB_UDI.LineC1.DownstreamAccu.Conveyor[_."Conveyor_C1.7.6"],
	                       Interlock := _.LineC1.DB_UDI.LineC1.Interlock.Conveyor[_."Conveyor_C1.7.6"]);
	    ;
	END_REGION
	
	
	REGION Conveyor_C1.7.7
	    #"Conveyor_C1.7.7"(ConveyorID := _."Conveyor_C1.7.7",
	                       Fault := _.LineC1.DB_UDI.LineC1.Fault.Conveyor[_."Conveyor_C1.7.7"],
	                       Upstream := _.LineC1.DB_UDI.LineC1.Upstream.Conveyor[_."Conveyor_C1.7.7"],
	                       Downstream := _.LineC1.DB_UDI.LineC1.DownstreamAccu.Conveyor[_."Conveyor_C1.7.7"],
	                       Interlock := _.LineC1.DB_UDI.LineC1.Interlock.Conveyor[_."Conveyor_C1.7.7"]);
	    ;
	END_REGION
	
	
	REGION "Conveyor_C1.7.8
	    #"Conveyor_C1.7.8"(ConveyorID := _."Conveyor_C1.7.8",
	                       Fault := _.LineC1.DB_UDI.LineC1.Fault.Conveyor[_."Conveyor_C1.7.8"],
	                       Upstream := _.LineC1.DB_UDI.LineC1.Upstream.Conveyor[_."Conveyor_C1.7.8"],
	                       Downstream := _.LineC1.DB_UDI.LineC1.DownstreamAccu.Conveyor[_."Conveyor_C1.7.8"],
	                       Interlock := _.LineC1.DB_UDI.LineC1.Interlock.Conveyor[_."Conveyor_C1.7.8"]);
	    ;
	END_REGION
	
	
	REGION Conveyor_C1.7.9
	    #"Conveyor_C1.7.9"(ConveyorID := _."Conveyor_C1.7.9",
	                       Fault := _.LineC1.DB_UDI.LineC1.Fault.Conveyor[_."Conveyor_C1.7.9"],
	                       Upstream := _.LineC1.DB_UDI.LineC1.Upstream.Conveyor[_."Conveyor_C1.7.9"],
	                       Downstream := _.LineC1.DB_UDI.LineC1.DownstreamAccu.Conveyor[_."Conveyor_C1.7.9"],
	                       Interlock := _.LineC1.DB_UDI.LineC1.Interlock.Conveyor[_."Conveyor_C1.7.9"]);
	    ;
	END_REGION
	
	
	REGION Conveyor_C1.7.10
	    #"Conveyor_C1.7.10"(ConveyorID := _."Conveyor_C1.7.10",
	                        Fault := _.LineC1.DB_UDI.LineC1.Fault.Conveyor[_."Conveyor_C1.7.10"],
	                        Upstream := _.LineC1.DB_UDI.LineC1.Upstream.Conveyor[_."Conveyor_C1.7.10"],
	                        Downstream := _.LineC1.DB_UDI.LineC1.DownstreamAccu.Conveyor[_."Conveyor_C1.7.10"],
	                        Interlock := _.LineC1.DB_UDI.LineC1.Interlock.Conveyor[_."Conveyor_C1.7.10"]);
	    ;
	END_REGION
	
	
	
	REGION Conveyor_C1.9.1
	    #"Conveyor_C1.9.1"(ConveyorID := _."Conveyor_C1.9.1",
	                       Fault := _.LineC1.DB_UDI.LineC1.Fault.Conveyor[_."Conveyor_C1.9.1"],
	                       Upstream := _.LineC1.DB_UDI.LineC1.Upstream.Conveyor[_."Conveyor_C1.9.1"],
	                       Downstream := _.LineC1.DB_UDI.LineC1.DownstreamAccu.Conveyor[_."Conveyor_C1.9.1"],
	                       Interlock := _.LineC1.DB_UDI.LineC1.Interlock.Conveyor[_."Conveyor_C1.9.1"]);
	    ;
	END_REGION
	
	
	REGION Conveyor_C1.10.1
	    #"Conveyor_C1.10.1"(ConveyorID := _."Conveyor_C1.10.1",
	                        Fault := _.LineC1.DB_UDI.LineC1.Fault.Conveyor[_."Conveyor_C1.10.1"],
	                        Upstream := _.LineC1.DB_UDI.LineC1.Upstream.Conveyor[_."Conveyor_C1.10.1"],
	                        Downstream := _.LineC1.DB_UDI.LineC1.DownstreamAccu.Conveyor[_."Conveyor_C1.10.1"],
	                        Interlock := _.LineC1.DB_UDI.LineC1.Interlock.Conveyor[_."Conveyor_C1.10.1"]);
	    ;
	END_REGION
	
	
	REGION Conveyor_C1.11.1
	    #"Conveyor_C1.11.1"(ConveyorID := _."Conveyor_C1.11.1",
	                        Fault := _.LineC1.DB_UDI.LineC1.Fault.Conveyor[_."Conveyor_C1.11.1"],
	                        Upstream := _.LineC1.DB_UDI.LineC1.Upstream.Conveyor[_."Conveyor_C1.11.1"],
	                        Downstream := _.LineC1.DB_UDI.LineC1.DownstreamAccu.Conveyor[_."Conveyor_C1.11.1"],
	                        Interlock := _.LineC1.DB_UDI.LineC1.Interlock.Conveyor[_."Conveyor_C1.11.1"]);
	    ;
	END_REGION
	
	
	REGION Conveyor_C1.11.2
	    #"Conveyor_C1.11.2"(ConveyorID := _."Conveyor_C1.11.2",
	                        Fault := _.LineC1.DB_UDI.LineC1.Fault.Conveyor[_."Conveyor_C1.11.2"],
	                        Upstream := _.LineC1.DB_UDI.LineC1.Upstream.Conveyor[_."Conveyor_C1.11.2"],
	                        Downstream := _.LineC1.DB_UDI.LineC1.DownstreamAccu.Conveyor[_."Conveyor_C1.11.2"],
	                        Interlock := _.LineC1.DB_UDI.LineC1.Interlock.Conveyor[_."Conveyor_C1.11.2"]);
	    ;
	END_REGION
	
	
	REGION Conveyor_C1.12.1
	    #"Conveyor_C1.12.1"(ConveyorID := _."Conveyor_C1.12.1",
	                        Fault := _.LineC1.DB_UDI.LineC1.Fault.Conveyor[_."Conveyor_C1.12.1"],
	                        Upstream := _.LineC1.DB_UDI.LineC1.Upstream.Conveyor[_."Conveyor_C1.12.1"],
	                        Downstream := _.LineC1.DB_UDI.LineC1.DownstreamAccu.Conveyor[_."Conveyor_C1.12.1"],
	                        Interlock := _.LineC1.DB_UDI.LineC1.Interlock.Conveyor[_."Conveyor_C1.12.1"]);
	    ;
	END_REGION
	
	
	REGION Conveyor_C1.12.2
	    #"Conveyor_C1.12.2"(ConveyorID := _."Conveyor_C1.12.2",
	                        Fault := _.LineC1.DB_UDI.LineC1.Fault.Conveyor[_."Conveyor_C1.12.2"],
	                        Upstream := _.LineC1.DB_UDI.LineC1.Upstream.Conveyor[_."Conveyor_C1.12.2"],
	                        Downstream := _.LineC1.DB_UDI.LineC1.DownstreamAccu.Conveyor[_."Conveyor_C1.12.2"],
	                        Interlock := _.LineC1.DB_UDI.LineC1.Interlock.Conveyor[_."Conveyor_C1.12.2"]);
	    ;
	END_REGION
	
	
	REGION Conveyor_C1.12.3
	    #"Conveyor_C1.12.3"(ConveyorID := _."Conveyor_C1.12.3",
	                        Fault := _.LineC1.DB_UDI.LineC1.Fault.Conveyor[_."Conveyor_C1.12.3"],
	                        Upstream := _.LineC1.DB_UDI.LineC1.Upstream.Conveyor[_."Conveyor_C1.12.3"],
	                        Downstream := _.LineC1.DB_UDI.LineC1.DownstreamAccu.Conveyor[_."Conveyor_C1.12.3"],
	                        Interlock := _.LineC1.DB_UDI.LineC1.Interlock.Conveyor[_."Conveyor_C1.12.3"]);
	    ;
	END_REGION
	
	
	REGION Transfer_C1.13.1
	    #"Transfer_C1.13.1"(TransferID:=_."Transfer_C1.13.1",
	                        Fault:=_.LineC1.DB_UDI.LineC1.Fault.Conveyor[_."Transfer_C1.13.1"],
	                        Upstream:=_.LineC1.DB_UDI.LineC1.Upstream.Conveyor[_."Transfer_C1.13.1"],
	                        Downstream:=_.LineC1.DB_UDI.LineC1.DownstreamAccu.Conveyor[_."Transfer_C1.13.1"],
	                        FrontSensorFilterTime:=_.LineC1.DB_ConveyorParameters.Line.C1.Transfer[_."Transfer_C1.13.1"].setTransferTimer,
	                        TransferDirection:=_.Global.DB_ToteTracking.Conveyor[_."Transfer_C1.13.1"].ToteDir);
	    
	END_REGION
	
	
	REGION Transfer_C1.14.1
	    #"Transfer_C1.14.1"(TransferID := _."Transfer_C1.14.1",
	                        Fault := _.LineC1.DB_UDI.LineC1.Fault.Conveyor[_."Transfer_C1.14.1"],
	                        Upstream := _.LineC1.DB_UDI.LineC1.Upstream.Conveyor[_."Transfer_C1.14.1"],
	                        Downstream := _.LineC1.DB_UDI.LineC1.DownstreamAccu.Conveyor[_."Transfer_C1.14.1"],
	                        FrontSensorFilterTime := _.LineC1.DB_ConveyorParameters.Line.C1.Transfer[_."Transfer_C1.14.1"].setTransferTimer,
	                        TransferDirection := _.Global.DB_ToteTracking.Conveyor[_."Transfer_C1.14.1"].ToteDir);
	END_REGION
	
	
	REGION Conveyor_C1.15.2
	    #"Conveyor_C1.15.2"(ConveyorID := _."Conveyor_C1.15.2",
	                        Fault := _.LineC1.DB_UDI.LineC1.Fault.Conveyor[_."Conveyor_C1.15.2"],
	                        Upstream := _.LineC1.DB_UDI.LineC1.Upstream.Conveyor[_."Conveyor_C1.15.2"],
	                        Downstream := _.LineC1.DB_UDI.LineC1.DownstreamAccu.Conveyor[_."Conveyor_C1.15.2"],
	                        Interlock := _.LineC1.DB_UDI.LineC1.Interlock.Conveyor[_."Conveyor_C1.15.2"]);
	    ;
	END_REGION
	
	
	REGION Conveyor_C1.15.3
	    #"Conveyor_C1.15.3"(ConveyorID := _."Conveyor_C1.15.3",
	                        Fault := _.LineC1.DB_UDI.LineC1.Fault.Conveyor[_."Conveyor_C1.15.3"],
	                        Upstream := _.LineC1.DB_UDI.LineC1.Upstream.Conveyor[_."Conveyor_C1.15.3"],
	                        Downstream := _.LineC1.DB_UDI.LineC1.DownstreamAccu.Conveyor[_."Conveyor_C1.15.3"],
	                        Interlock := _.LineC1.DB_UDI.LineC1.Interlock.Conveyor[_."Conveyor_C1.15.3"]);
	    ;
	END_REGION
	
	
	REGION Conveyor_C1.15.4
	    #"Conveyor_C1.15.4"(ConveyorID := _."Conveyor_C1.15.4",
	                        Fault := _.LineC1.DB_UDI.LineC1.Fault.Conveyor[_."Conveyor_C1.15.4"],
	                        Upstream := _.LineC1.DB_UDI.LineC1.Upstream.Conveyor[_."Conveyor_C1.15.4"],
	                        Downstream := _.LineC1.DB_UDI.LineC1.DownstreamAccu.Conveyor[_."Conveyor_C1.15.4"],
	                        Interlock := _.LineC1.DB_UDI.LineC1.Interlock.Conveyor[_."Conveyor_C1.15.4"]);
	    ;
	END_REGION
	
	
	REGION Conveyor_C1.16.1
	    #"Conveyor_C1.16.1"(ConveyorID := _."Conveyor_C1.16.1",
	                        Fault := _.LineC1.DB_UDI.LineC1.Fault.Conveyor[_."Conveyor_C1.16.1"],
	                        Upstream := _.LineC1.DB_UDI.LineC1.Upstream.Conveyor[_."Conveyor_C1.16.1"],
	                        Downstream := _.LineC1.DB_UDI.LineC1.DownstreamAccu.Conveyor[_."Conveyor_C1.16.1"],
	                        Interlock := _.LineC1.DB_UDI.LineC1.Interlock.Conveyor[_."Conveyor_C1.16.1"]);
	    ;
	END_REGION
	
	
	REGION Conveyor_C1.18.1
	    #"Conveyor_C1.18.1"(ConveyorID := _."Conveyor_C1.18.1",
	                        Fault := _.LineC1.DB_UDI.LineC1.Fault.Conveyor[_."Conveyor_C1.18.1"],
	                        Upstream := _.LineC1.DB_UDI.LineC1.Upstream.Conveyor[_."Conveyor_C1.18.1"],
	                        Downstream := _.LineC1.DB_UDI.LineC1.DownstreamAccu.Conveyor[_."Conveyor_C1.18.1"],
	                        Interlock := _.LineC1.DB_UDI.LineC1.Interlock.Conveyor[_."Conveyor_C1.18.1"]);
	    ;
	END_REGION
	
	
	REGION Conveyor_C1.18.2
	    #"Conveyor_C1.18.2"(ConveyorID := _."Conveyor_C1.18.2",
	                        Fault := _.LineC1.DB_UDI.LineC1.Fault.Conveyor[_."Conveyor_C1.18.2"],
	                        Upstream := _.LineC1.DB_UDI.LineC1.Upstream.Conveyor[_."Conveyor_C1.18.2"],
	                        Downstream := _.LineC1.DB_UDI.LineC1.DownstreamAccu.Conveyor[_."Conveyor_C1.18.2"],
	                        Interlock := _.LineC1.DB_UDI.LineC1.Interlock.Conveyor[_."Conveyor_C1.18.2"]);
	    ;
	END_REGION
	
	
	REGION Conveyor_C1.18.3
	    #"Conveyor_C1.18.3"(ConveyorID := _."Conveyor_C1.18.3",
	                        Fault := _.LineC1.DB_UDI.LineC1.Fault.Conveyor[_."Conveyor_C1.18.3"],
	                        Upstream := _.LineC1.DB_UDI.LineC1.Upstream.Conveyor[_."Conveyor_C1.18.3"],
	                        Downstream := _.LineC1.DB_UDI.LineC1.DownstreamAccu.Conveyor[_."Conveyor_C1.18.3"],
	                        Interlock := _.LineC1.DB_UDI.LineC1.Interlock.Conveyor[_."Conveyor_C1.18.3"]);
	    ;
	END_REGION
	
	
	REGION Conveyor_C1.18.4
	    #"Conveyor_C1.18.4"(ConveyorID := _."Conveyor_C1.18.4",
	                        Fault := _.LineC1.DB_UDI.LineC1.Fault.Conveyor[_."Conveyor_C1.18.4"],
	                        Upstream := _.LineC1.DB_UDI.LineC1.Upstream.Conveyor[_."Conveyor_C1.18.4"],
	                        Downstream := _.LineC1.DB_UDI.LineC1.DownstreamAccu.Conveyor[_."Conveyor_C1.18.4"],
	                        Interlock := _.LineC1.DB_UDI.LineC1.Interlock.Conveyor[_."Conveyor_C1.18.4"]);
	    ;
	END_REGION
	
	
	REGION Conveyor_C1.18.5
	    #"Conveyor_C1.18.5"(ConveyorID := _."Conveyor_C1.18.5",
	                        Fault := _.LineC1.DB_UDI.LineC1.Fault.Conveyor[_."Conveyor_C1.18.5"],
	                        Upstream := _.LineC1.DB_UDI.LineC1.Upstream.Conveyor[_."Conveyor_C1.18.5"],
	                        Downstream := _.LineC1.DB_UDI.LineC1.DownstreamAccu.Conveyor[_."Conveyor_C1.18.5"],
	                        Interlock := _.LineC1.DB_UDI.LineC1.Interlock.Conveyor[_."Conveyor_C1.18.5"]);
	    ;
	END_REGION
	
	
	REGION Conveyor_C1.18.6
	    #"Conveyor_C1.18.6"(ConveyorID := _."Conveyor_C1.18.6",
	                        Fault := _.LineC1.DB_UDI.LineC1.Fault.Conveyor[_."Conveyor_C1.18.6"],
	                        Upstream := _.LineC1.DB_UDI.LineC1.Upstream.Conveyor[_."Conveyor_C1.18.6"],
	                        Downstream := _.LineC1.DB_UDI.LineC1.DownstreamAccu.Conveyor[_."Conveyor_C1.18.6"],
	                        Interlock := _.LineC1.DB_UDI.LineC1.Interlock.Conveyor[_."Conveyor_C1.18.6"]);
	    ;
	END_REGION
	
	
	REGION Conveyor_C1.18.7
	    #"Conveyor_C1.18.7"(ConveyorID := _."Conveyor_C1.18.7",
	                        Fault := _.LineC1.DB_UDI.LineC1.Fault.Conveyor[_."Conveyor_C1.18.7"],
	                        Upstream := _.LineC1.DB_UDI.LineC1.Upstream.Conveyor[_."Conveyor_C1.18.7"],
	                        Downstream := _.LineC1.DB_UDI.LineC1.DownstreamAccu.Conveyor[_."Conveyor_C1.18.7"],
	                        Interlock := _.LineC1.DB_UDI.LineC1.Interlock.Conveyor[_."Conveyor_C1.18.7"]);
	    ;
	END_REGION
	
	
	REGION Conveyor_C1.19.1
	    #"Conveyor_C1.19.1"(ConveyorID := _."Conveyor_C1.19.1",
	                        Fault := _.LineC1.DB_UDI.LineC1.Fault.Conveyor[_."Conveyor_C1.19.1"],
	                        Upstream := _.LineC1.DB_UDI.LineC1.Upstream.Conveyor[_."Conveyor_C1.19.1"],
	                        Downstream := _.LineC1.DB_UDI.LineC1.DownstreamAccu.Conveyor[_."Conveyor_C1.19.1"],
	                        Interlock := _.LineC1.DB_UDI.LineC1.Interlock.Conveyor[_."Conveyor_C1.19.1"]);
	    ;
	END_REGION
	
	
	REGION Conveyor_C1.20.2
	    #"Conveyor_C1.20.2"(ConveyorID := _."Conveyor_C1.20.2",
	                        Fault := _.LineC1.DB_UDI.LineC1.Fault.Conveyor[_."Conveyor_C1.20.2"],
	                        Upstream := _.LineC1.DB_UDI.LineC1.Upstream.Conveyor[_."Conveyor_C1.20.2"],
	                        Downstream := _.LineC1.DB_UDI.LineC1.DownstreamAccu.Conveyor[_."Conveyor_C1.20.2"],
	                        Interlock := _.LineC1.DB_UDI.LineC1.Interlock.Conveyor[_."Conveyor_C1.20.2"]);
	    ;
	END_REGION
	
	
	
	
	
	
	
	
END_FUNCTION_BLOCK
END_NAMESPACE

NAMESPACE LineC1
ORGANIZATION_BLOCK Main_LineC1
TITLE = "Main Program Sweep (Cycle)"
{ S7_Optimized_Access := 'TRUE' ; Published := 'FALSE' }
VERSION : 0.1

BEGIN
	// ==========================================================================================================================================
	// Company        : LogTech, s.r.o.
	// Created by     : Mahmoud Elnady
	// Block          : FC_UpstreaProductionTote
	// Project        : Lekarna, Chrudim -PLC001 -MCC001
	// Project number : 23-157
	// ==========================================================================================================================================
	
	
	IDB_LineC1();
	
	FC_Upstream();
	
	FC_Downstream();
	
	IDB_FB_Merging();
	
END_ORGANIZATION_BLOCK
END_NAMESPACE

NAMESPACE LineD1
FUNCTION_BLOCK FB_LineD1
{ S7_Optimized_Access := 'TRUE' ; Published := 'TRUE' }
VERSION : 0.1
   VAR 
      "Conveyor_D1.1.1" { S7_SetPoint := 'False'} : _.Global.FB_Conveyor;
      "MABS_D1.1.1" { S7_SetPoint := 'False'} : _.Global.FB_MABS;
      "Transfer_D1.1.1" { S7_SetPoint := 'False'} : _.Global.FB_S300_tTransMode;
   END_VAR


BEGIN
	
	
	
	
	
	
	
	
	
	
	
	
	
	
	
END_FUNCTION_BLOCK
END_NAMESPACE

NAMESPACE LineD1
ORGANIZATION_BLOCK Main_LineD1
TITLE = "Main Program Sweep (Cycle)"
{ S7_Optimized_Access := 'TRUE' ; Published := 'FALSE' }
VERSION : 0.1

BEGIN
	IDB_LineD1();
	
END_ORGANIZATION_BLOCK
END_NAMESPACE

NAMESPACE EmptyLine
FUNCTION_BLOCK FB_EmptyLine
{ S7_Optimized_Access := 'TRUE' ; Published := 'TRUE' }
VERSION : 0.1
   VAR 
      "J1.1.1" { S7_SetPoint := 'False'} : _.Global.FB_Conveyor;
      "J1.1.2" : _.Global.FB_Conveyor;
      "J1.1.3" : _.Global.FB_Conveyor;
      "J1.1.4" : _.Global.FB_Conveyor;
      "J1.1.5" : _.Global.FB_Conveyor;
      "J1.1.6" : _.Global.FB_Conveyor;
      "J1.1.7" : _.Global.FB_Conveyor;
      "J1.1.8" : _.Global.FB_Conveyor;
      "J1.1.9" : _.Global.FB_Conveyor;
      "J1.1.10" : _.Global.FB_Conveyor;
      "J1.1.11" : _.Global.FB_Conveyor;
      "J1.1.12" : _.Global.FB_Conveyor;
      "J1.1.13" : _.Global.FB_Conveyor;
      "J1.1.14" : _.Global.FB_Conveyor;
      "J1.1.15" : _.Global.FB_Conveyor;
      "J1.1.16" : _.Global.FB_Conveyor;
      "J1.2.1" : _.Global.FB_Conveyor;
      "J1.2.2" : _.Global.FB_Conveyor;
      "J1.2.3" : _.Global.FB_Conveyor;
      "J2.1.1" : _.Global.FB_Conveyor;
      "J2.1.2" : _.Global.FB_Conveyor;
      "J2.1.3" : _.Global.FB_Conveyor;
      "J2.1.4" : _.Global.FB_Conveyor;
      "J2.1.5" : _.Global.FB_Conveyor;
      "J2.1.6" : _.Global.FB_Conveyor;
      "J2.1.7" : _.Global.FB_Conveyor;
      "J2.1.8" : _.Global.FB_Conveyor;
      "J2.1.9" : _.Global.FB_Conveyor;
      "J2.1.10" : _.Global.FB_Conveyor;
      "J2.1.11" : _.Global.FB_Conveyor;
      "J2.1.12" : _.Global.FB_Conveyor;
      "J2.1.13" : _.Global.FB_Conveyor;
      "J2.1.14" : _.Global.FB_Conveyor;
      "J2.1.15" : _.Global.FB_Conveyor;
      "J2.2.1" : _.Global.FB_Conveyor;
      "J2.2.2" : _.Global.FB_Conveyor;
      "J2.3.1" : _.Global.FB_Conveyor;
      "J2.4.1" : _.Global.FB_Conveyor;
      "J1.2.4" : _.Global.FB_Conveyor;
      "J1.2.5" : _.Global.FB_Conveyor;
      "J1.3.1" : _.Global.FB_Conveyor;
      "J1.3.2" : _.Global.FB_Conveyor;
      "J1.4.1" : _.Global.FB_Conveyor;
      "J1.4.2" : _.Global.FB_Conveyor;
      "J1.4.3" : _.Global.FB_Conveyor;
      "J1.4.4" : _.Global.FB_Conveyor;
      "J1.4.5" : _.Global.FB_Conveyor;
      "J1.4.6" : _.Global.FB_Conveyor;
      "J1.4.7" : _.Global.FB_Conveyor;
      "J1.5.1" : _.Global.FB_Conveyor;
      "J1.5.2" : _.Global.FB_Conveyor;
      "J1.5.3" : _.Global.FB_Conveyor;
      "J1.5.4" : _.Global.FB_Conveyor;
      "J1.6.1" : _.Global.FB_MABS;
      "J1.6.2" : _.Global.FB_MABS;
      "J1.7.1" : _.Global.FB_Conveyor;
      "J1.7.2" : _.Global.FB_Conveyor;
      "J1.8.1" : _.Global.FB_Conveyor;
      "J1.8.2" : _.Global.FB_Conveyor;
      "J1.9.1" : _.Global.FB_Conveyor;
      "J1.10.1" : _.Global.FB_Conveyor;
      "J1.11.1" : _.Global.FB_Conveyor;
      "J1.11.2" : _.Global.FB_Conveyor;
      "J1.11.3" : _.Global.FB_Conveyor;
      "J1.11.4" : _.Global.FB_Conveyor;
      "J1.11.5" : _.Global.FB_Conveyor;
      "J1.11.6" : _.Global.FB_Conveyor;
      "J1.11.7" : _.Global.FB_Conveyor;
      "J1.11.8" : _.Global.FB_Conveyor;
      "J1.11.9" : _.Global.FB_Conveyor;
      "J1.11.10" : _.Global.FB_Conveyor;
      "J1.11.11" : _.Global.FB_Conveyor;
      "J1.11.12" : _.Global.FB_Conveyor;
      "J1.11.13" : _.Global.FB_Conveyor;
      "K1.1.1" : _.Global.FB_Conveyor;
      "K1.2.1" : _.Global.FB_Conveyor;
      "K1.3.1" : _.Global.FB_Conveyor;
      "K1.4.1" : _.Global.FB_Conveyor;
      "K1.4.2" : _.Global.FB_Conveyor;
      "K1.4.3" : _.Global.FB_Conveyor;
      "K1.4.4" : _.Global.FB_Conveyor;
      "K1.4.5" : _.Global.FB_Conveyor;
      "K1.4.6" : _.Global.FB_Conveyor;
      "K1.4.7" : _.Global.FB_Conveyor;
      "K1.4.8" : _.Global.FB_Conveyor;
      "K1.4.9" : _.Global.FB_Conveyor;
      "K1.4.10" : _.Global.FB_Conveyor;
      "K1.5.1" : _.Global.FB_Conveyor;
      "K1.5.2" : _.Global.FB_Conveyor;
      "K1.5.3" : _.Global.FB_Conveyor;
      "K1.5.4" : _.Global.FB_Conveyor;
      "K1.5.5" : _.Global.FB_Conveyor;
      "K1.5.6" : _.Global.FB_Conveyor;
      "K1.5.7" : _.Global.FB_Conveyor;
      "K1.5.8" : _.Global.FB_Conveyor;
      "K1.6.1" : _.Global.FB_Conveyor;
      "K1.6.2" : _.Global.FB_Conveyor;
      "K1.7.1" : _.Global.FB_Conveyor;
      "K1.7.2" : _.Global.FB_Conveyor;
      "K1.8.1" : _.Global.FB_Conveyor;
      "K1.8.2" : _.Global.FB_Conveyor;
      "K1.8.3" : _.Global.FB_Conveyor;
      "K1.9.1" : _.Global.FB_Conveyor;
      "K1.9.2" : _.Global.FB_Conveyor;
      "K1.9.3" : _.Global.FB_Conveyor;
      "K1.9.4" : _.Global.FB_Conveyor;
      "K1.9.5" : _.Global.FB_Conveyor;
      "K1.9.6" : _.Global.FB_Conveyor;
      "K1.9.7" : _.Global.FB_Conveyor;
      "K1.10.1" : _.Global.FB_Conveyor;
   END_VAR


BEGIN
	// ==========================================================================================================================================
	// Company        : LogTech, s.r.o.
	// Created by     : Anton Vinoth Soundraraj
	// Block          : FB_LineB1
	// Project        : Lékarna DC Chrudim
	// Project number : 23-157
	// ==========================================================================================================================================
	
	REGION J1.1.1
	    //J1.1.1
	    #"J1.1.1"(ConveyorID:=_."J1.1.1",
	              ConveyorSensor:=_."ASiGW-MCC001-bw143-C1: Input"."Sensor J1.1.1",
	                   Fault:= DB_UDI.EmptyLine.Fault.Stop.Conveyor[_."J1.1.1"],
	                   Upstream:= DB_UDI.EmptyLine.Upstream.Conveyor[_."J1.1.1"],
	                   Downstream:= DB_UDI.EmptyLine.DownstreamAcu.Stop.Conveyor[_."J1.1.1"],
	                   Interlock:= DB_UDI.EmptyLine.Interlock.Stop.Conveyor[_."J1.1.1"],
	                   RunForward=>_."ASiGW-MCC001-bw143-C1: Output"."Motor J1.1.1",
	                   WriteAsiDir=>_."ASiGW-MCC001-bw143-C1: Output"."Dir J1.1.1");
	
	END_REGION
	
	REGION J1.1.2
	    //J1.1.2
	    #"J1.1.2"(ConveyorID:=_."J1.1.2",
	              ConveyorSensor:=_."ASiGW-MCC001-bw143-C1: Input"."Sensor J1.1.2",
	                   Fault:= DB_UDI.EmptyLine.Fault.Stop.Conveyor[_."J1.1.2"],
	                   Upstream:= DB_UDI.EmptyLine.Upstream.Conveyor[_."J1.1.2"],
	                   Downstream:= DB_UDI.EmptyLine.DownstreamAcu.Stop.Conveyor[_."J1.1.2"],
	                   Interlock:= DB_UDI.EmptyLine.Interlock.Stop.Conveyor[_."J1.1.2"],
	                   RunForward=>_."ASiGW-MCC001-bw143-C1: Output"."Motor J1.1.2",
	                   WriteAsiDir=>_."ASiGW-MCC001-bw143-C1: Output"."Dir J1.1.2");
	
	END_REGION
	
	REGION J1.1.3
	    //J1.1.3
	    #"J1.1.3"(ConveyorID:=_."J1.1.3",
	              ConveyorSensor:=_."ASiGW-MCC001-bw143-C1: Input"."Sensor J1.1.11",
	                   Fault:= DB_UDI.EmptyLine.Fault.Stop.Conveyor[_."J1.1.3"],
	                   Upstream:= DB_UDI.EmptyLine.Upstream.Conveyor[_."J1.1.3"],
	                   Downstream:= DB_UDI.EmptyLine.DownstreamAcu.Stop.Conveyor[_."J1.1.3"],
	                   Interlock:= DB_UDI.EmptyLine.Interlock.Stop.Conveyor[_."J1.1.3"],
	                   RunForward=>_."ASiGW-MCC001-bw143-C1: Output"."Motor J1.1.3",
	                   WriteAsiDir=>_."ASiGW-MCC001-bw143-C1: Output"."Dir J1.1.3");
	     END_REGION
	
	REGION J1.1.4
	    //J1.1.4
	    #"J1.1.4"(ConveyorID:=_."J1.1.4",
	              ConveyorSensor:=_."ASiGW-MCC001-bw143-C1: Input"."Sensor J1.1.11",
	                   Fault:= DB_UDI.EmptyLine.Fault.Stop.Conveyor[_."J1.1.4"],
	                   Upstream:= DB_UDI.EmptyLine.Upstream.Conveyor[_."J1.1.4"],
	                   Downstream:= DB_UDI.EmptyLine.DownstreamAcu.Stop.Conveyor[_."J1.1.4"],
	                   Interlock:= DB_UDI.EmptyLine.Interlock.Stop.Conveyor[_."J1.1.4"],
	                   RunForward=>_."ASiGW-MCC001-bw143-C1: Output"."Motor J1.1.4",
	                   WriteAsiDir=>_."ASiGW-MCC001-bw143-C1: Output"."Dir J1.1.4");
	
	END_REGION
	
	REGION J1.1.5
	    //J1.1.5
	    #"J1.1.5"(ConveyorID := _."J1.1.5",
	              ConveyorSensor:=_."ASiGW-MCC001-bw143-C1: Input"."Sensor J1.1.11",
	              Fault := DB_UDI.EmptyLine.Fault.Stop.Conveyor[_."J1.1.5"],
	              Upstream := DB_UDI.EmptyLine.Upstream.Conveyor[_."J1.1.5"],
	              Downstream := DB_UDI.EmptyLine.DownstreamAcu.Stop.Conveyor[_."J1.1.5"],
	              Interlock := DB_UDI.EmptyLine.Interlock.Stop.Conveyor[_."J1.1.5"],
	              RunForward => _."ASiGW-MCC001-bw143-C1: Output"."Motor J1.1.5",
	              WriteAsiDir => _."ASiGW-MCC001-bw143-C1: Output"."Dir J1.1.5");
	END_REGION
	
	REGION J1.1.6
	    //J1.1.6
	    #"J1.1.6"(ConveyorID := _."J1.1.6",
	              ConveyorSensor:=_."ASiGW-MCC001-bw143-C1: Input"."Sensor J1.1.11",
	              Fault := DB_UDI.EmptyLine.Fault.Stop.Conveyor[_."J1.1.6"],
	              Upstream := DB_UDI.EmptyLine.Upstream.Conveyor[_."J1.1.6"],
	              Downstream := DB_UDI.EmptyLine.DownstreamAcu.Stop.Conveyor[_."J1.1.6"],
	              Interlock := DB_UDI.EmptyLine.Interlock.Stop.Conveyor[_."J1.1.6"],
	              RunForward => _."ASiGW-MCC001-bw143-C1: Output"."Motor J1.1.6",
	              WriteAsiDir => _."ASiGW-MCC001-bw143-C1: Output"."Dir J1.1.6");
	    
	END_REGION
	
	REGION J1.1.7
	    //J1.1.7
	    #"J1.1.7"(ConveyorID := _."J1.1.7",
	              ConveyorSensor:=_."ASiGW-MCC001-bw143-C1: Input"."Sensor J1.1.11",
	              Fault := DB_UDI.EmptyLine.Fault.Stop.Conveyor[_."J1.1.7"],
	              Upstream := DB_UDI.EmptyLine.Upstream.Conveyor[_."J1.1.7"],
	              Downstream := DB_UDI.EmptyLine.DownstreamAcu.Stop.Conveyor[_."J1.1.7"],
	              Interlock := DB_UDI.EmptyLine.Interlock.Stop.Conveyor[_."J1.1.7"],
	              RunForward => _."ASiGW-MCC001-bw143-C1: Output"."Motor J1.1.7",
	              WriteAsiDir => _."ASiGW-MCC001-bw143-C1: Output"."Dir J1.1.7");
	    
	END_REGION
	
	REGION J1.1.8
	    //J1.1.8
	    #"J1.1.8"(ConveyorID := _."J1.1.8",
	              ConveyorSensor:=_."ASiGW-MCC001-bw143-C1: Input"."Sensor J1.1.11",
	              Fault := DB_UDI.EmptyLine.Fault.Stop.Conveyor[_."J1.1.8"],
	              Upstream := DB_UDI.EmptyLine.Upstream.Conveyor[_."J1.1.8"],
	              Downstream := DB_UDI.EmptyLine.DownstreamAcu.Stop.Conveyor[_."J1.1.8"],
	              Interlock := DB_UDI.EmptyLine.Interlock.Stop.Conveyor[_."J1.1.8"],
	              RunForward=>_."ASiGW-MCC001-bw143-C1: Output"."Motor J1.1.8",
	              WriteAsiDir=>_."ASiGW-MCC001-bw143-C1: Output"."Dir J1.1.8");
	    
	END_REGION
	
	REGION J1.1.9
	    //J1.1.9
	    #"J1.1.9"(ConveyorID := _."J1.1.9",
	              ConveyorSensor:=_."ASiGW-MCC001-bw143-C1: Input"."Sensor J1.1.11",
	              Fault := DB_UDI.EmptyLine.Fault.Stop.Conveyor[_."J1.1.9"],
	              Upstream := DB_UDI.EmptyLine.Upstream.Conveyor[_."J1.1.9"],
	              Downstream := DB_UDI.EmptyLine.DownstreamAcu.Stop.Conveyor[_."J1.1.9"],
	              Interlock := DB_UDI.EmptyLine.Interlock.Stop.Conveyor[_."J1.1.9"],
	              RunForward=>_."ASiGW-MCC001-bw143-C1: Output"."Motor J1.1.9",
	              WriteAsiDir=>_."ASiGW-MCC001-bw143-C1: Output"."Dir J1.1.9");
	END_REGION
	
	REGION J1.1.10
	    //J1.1.10
	    #"J1.1.10"(ConveyorID := _."J1.1.10",
	               ConveyorSensor:=_."ASiGW-MCC001-bw143-C1: Input"."Sensor J1.1.11",
	               Fault := DB_UDI.EmptyLine.Fault.Stop.Conveyor[_."J1.1.10"],
	               Upstream := DB_UDI.EmptyLine.Upstream.Conveyor[_."J1.1.10"],
	               Downstream := DB_UDI.EmptyLine.DownstreamAcu.Stop.Conveyor[_."J1.1.10"],
	               Interlock := DB_UDI.EmptyLine.Interlock.Stop.Conveyor[_."J1.1.10"],
	               RunForward=>_."ASiGW-MCC001-bw143-C1: Output"."Motor J1.1.10",
	               WriteAsiDir=>_."ASiGW-MCC001-bw143-C1: Output"."Dir J1.1.10");
	    
	END_REGION
	
	REGION J1.1.11
	    //J1.1.11
	    #"J1.1.11"(ConveyorID := _."J1.1.11",
	               ConveyorSensor:=_."ASiGW-MCC001-bw143-C1: Input"."Sensor J1.1.11",
	               Fault := DB_UDI.EmptyLine.Fault.Stop.Conveyor[_."J1.1.11"],
	               Upstream := DB_UDI.EmptyLine.Upstream.Conveyor[_."J1.1.11"],
	               Downstream := DB_UDI.EmptyLine.DownstreamAcu.Stop.Conveyor[_."J1.1.11"],
	               Interlock := DB_UDI.EmptyLine.Interlock.Stop.Conveyor[_."J1.1.11"],
	               RunForward=>_."ASiGW-MCC001-bw143-C1: Output"."Motor J1.1.11",
	               WriteAsiDir=>_."ASiGW-MCC001-bw143-C1: Output"."Dir J1.1.11");
	    
	END_REGION
	
	REGION J1.1.12
	    //J1.1.12
	    #"J1.1.12"(ConveyorID := _."J1.1.12",
	               ConveyorSensor:=_."ASiGW-MCC001-bw143-C1: Input"."Sensor J1.1.15",
	               Fault := DB_UDI.EmptyLine.Fault.Stop.Conveyor[_."J1.1.12"],
	               Upstream := DB_UDI.EmptyLine.Upstream.Conveyor[_."J1.1.12"],
	               Downstream := DB_UDI.EmptyLine.DownstreamAcu.Stop.Conveyor[_."J1.1.12"],
	               Interlock := DB_UDI.EmptyLine.Interlock.Stop.Conveyor[_."J1.1.12"],
	               RunForward=>_."ASiGW-MCC001-bw143-C1: Output"."Motor J1.1.12",
	               WriteAsiDir=>_."ASiGW-MCC001-bw143-C1: Output"."Dir J1.1.12");
	    
	END_REGION
	
	REGION J1.1.13
	    //J1.1.13
	    #"J1.1.13"(ConveyorID:=_."J1.1.13",
	               ConveyorSensor:=_."ASiGW-MCC001-bw143-C1: Input"."Sensor J1.1.15",
	               Fault:= DB_UDI.EmptyLine.Fault.Stop.Conveyor[_."J1.1.13"],
	               Upstream:= DB_UDI.EmptyLine.Upstream.Conveyor[_."J1.1.13"],
	               Downstream:= DB_UDI.EmptyLine.DownstreamAcu.Stop.Conveyor[_."J1.1.13"],
	               Interlock:= DB_UDI.EmptyLine.Interlock.Stop.Conveyor[_."J1.1.13"],
	               RunForward=>_."ASiGW-MCC001-bw143-C1: Output"."Motor J1.1.13",
	               WriteAsiDir=>_."ASiGW-MCC001-bw143-C1: Output"."Dir J1.1.13");
	        
	END_REGION
	
	REGION J1.1.14
	    //J1.1.14
	    #"J1.1.14"(ConveyorID:=_."J1.1.14",
	               ConveyorSensor:=_."ASiGW-MCC001-bw143-C1: Input"."Sensor J1.1.15",
	               Fault:= DB_UDI.EmptyLine.Fault.Stop.Conveyor[_."J1.1.14"],
	               Upstream:= DB_UDI.EmptyLine.Upstream.Conveyor[_."J1.1.14"],
	               Downstream:= DB_UDI.EmptyLine.DownstreamAcu.Stop.Conveyor[_."J1.1.14"],
	               Interlock:= DB_UDI.EmptyLine.Interlock.Stop.Conveyor[_."J1.1.14"],
	               RunForward=>_."ASiGW-MCC001-bw143-C1: Output"."Motor J1.1.14",
	               WriteAsiDir=>_."ASiGW-MCC001-bw143-C1: Output"."Dir J1.1.14");
	END_REGION
	
	REGION J1.1.15
	    //J1.1.15
	    #"J1.1.15"(ConveyorID:=_."J1.1.15",
	               ConveyorSensor:=_."ASiGW-MCC001-bw143-C1: Input"."Sensor J1.1.15",
	               Fault:= DB_UDI.EmptyLine.Fault.Stop.Conveyor[_."J1.1.15"],
	               Upstream:= DB_UDI.EmptyLine.Upstream.Conveyor[_."J1.1.15"],
	               Downstream:= DB_UDI.EmptyLine.DownstreamAcu.Stop.Conveyor[_."J1.1.15"],
	               Interlock:= DB_UDI.EmptyLine.Interlock.Stop.Conveyor[_."J1.1.15"],
	               RunForward=>_."ASiGW-MCC001-bw143-C1: Output"."Motor J1.1.15",
	               WriteAsiDir=>_."ASiGW-MCC001-bw143-C1: Output"."Dir J1.1.15");
	
	END_REGION
	
	REGION J1.2.1
	    //J1.2.1
	    #"J1.2.1"(ConveyorID := _."J1.2.1",
	              ConveyorSensor:=_."ASiGW-MCC001-bw143-C1: Input"."Sensor J1.2.1",
	              Fault := DB_UDI.EmptyLine.Fault.Stop.Conveyor[_."J1.2.1"],
	              Upstream := DB_UDI.EmptyLine.Upstream.Conveyor[_."J1.2.1"],
	              Downstream := DB_UDI.EmptyLine.DownstreamAcu.Stop.Conveyor[_."J1.2.1"],
	              Interlock := DB_UDI.EmptyLine.Interlock.Stop.Conveyor[_."J1.2.1"],
	              RunForward => _."ASiGW-MCC001-bw143-C1: Output"."Motor J1.2.1",
	              WriteAsiDir => _."ASiGW-MCC001-bw143-C1: Output"."Dir J1.2.1");
	    
	END_REGION
	
	REGION J1.2.2
	    //J1.2.2
	    #"J1.2.2"(ConveyorID:=_."J1.2.2",
	              ConveyorSensor:=_."ASiGW-MCC001-bw143-C1: Input"."Sensor J1.2.2",
	                   Fault:= DB_UDI.EmptyLine.Fault.Stop.Conveyor[_."J1.2.2"],
	                   Upstream:= DB_UDI.EmptyLine.Upstream.Conveyor[_."J1.2.2"],
	                   Downstream:= DB_UDI.EmptyLine.DownstreamAcu.Stop.Conveyor[_."J1.2.2"],
	                   Interlock:= DB_UDI.EmptyLine.Interlock.Stop.Conveyor[_."J1.2.2"],
	                   RunForward => _."ASiGW-MCC001-bw143-C1: Output"."Motor J1.2.2",
	                   WriteAsiDir => _."ASiGW-MCC001-bw143-C1: Output"."Dir J1.2.2");
	
	END_REGION
	
	REGION J1.2.3
	    //J1.2.3 Staright for Merger1
	    #"J1.2.3"(ConveyorID:=_."J1.2.3",
	              ConveyorSensor:=_."ASiGW-MCC001-bw143-C1: Input"."Sensor J1.2.3",
	                   Fault:= DB_UDI.EmptyLine.Fault.Stop.Conveyor[_."J1.2.3"],
	                   Upstream:= DB_UDI.EmptyLine.Upstream.Conveyor[_."J1.2.3"],
	                   Downstream:= DB_UDI.EmptyLine.DownstreamAcu.Stop.Conveyor[_."J1.2.3"],
	                   Interlock:= DB_UDI.EmptyLine.Interlock.Stop.Conveyor[_."J1.2.3"],
	                   RunForward => _."ASiGW-MCC001-bw143-C1: Output"."Motor J1.2.3",
	                   WriteAsiDir => _."ASiGW-MCC001-bw143-C1: Output"."Dir J1.2.3");
	
	END_REGION
	
	REGION J2.1.1
	    //J2.1.1
	    #"J2.1.1"(ConveyorID:=_."J2.1.1",
	              ConveyorSensor:=_."ASiGW-MCC001-bw200-C2: Input"."Sensor J2.1.1",
	                   Fault:= DB_UDI.EmptyLine.Fault.Stop.Conveyor[_."J2.1.1"],
	                   Upstream:= DB_UDI.EmptyLine.Upstream.Conveyor[_."J2.1.1"],
	                   Downstream:= DB_UDI.EmptyLine.DownstreamAcu.Stop.Conveyor[_."J2.1.1"],
	                   Interlock:= DB_UDI.EmptyLine.Interlock.Stop.Conveyor[_."J2.1.1"],
	                   RunForward=>_."ASiGW-MCC001-bw200-C2: Output"."Motor J2.1.1",
	                   WriteAsiDir=>_."ASiGW-MCC001-bw200-C2: Output"."Dir J2.1.1");
	
	END_REGION
	
	REGION J2.1.2
	    //J2.1.2
	    #"J2.1.2"(ConveyorID:=_."J2.1.2",
	              ConveyorSensor:=_."ASiGW-MCC001-bw200-C2: Input"."Sensor J2.1.2",
	                   Fault:= DB_UDI.EmptyLine.Fault.Stop.Conveyor[_."J2.1.2"],
	                   Upstream:= DB_UDI.EmptyLine.Upstream.Conveyor[_."J2.1.2"],
	                   Downstream:= DB_UDI.EmptyLine.DownstreamAcu.Stop.Conveyor[_."J2.1.2"],
	                   Interlock:= DB_UDI.EmptyLine.Interlock.Stop.Conveyor[_."J2.1.2"],
	                   RunForward=>_."ASiGW-MCC001-bw200-C2: Output"."Motor J2.1.2",
	                   WriteAsiDir=>_."ASiGW-MCC001-bw200-C2: Output"."Dir J2.1.2");
	
	END_REGION
	
	REGION J2.1.3
	    //J2.1.3
	    #"J2.1.3"(ConveyorID := _."J2.1.3",
	              ConveyorSensor:=_."ASiGW-MCC001-bw200-C2: Input"."Sensor J2.1.11",
	              Fault := DB_UDI.EmptyLine.Fault.Stop.Conveyor[_."J2.1.3"],
	              Upstream := DB_UDI.EmptyLine.Upstream.Conveyor[_."J2.1.3"],
	              Downstream := DB_UDI.EmptyLine.DownstreamAcu.Stop.Conveyor[_."J2.1.3"],
	              Interlock := DB_UDI.EmptyLine.Interlock.Stop.Conveyor[_."J2.1.3"],
	              RunForward => _."ASiGW-MCC001-bw200-C2: Output"."Motor J2.1.3",
	              WriteAsiDir => _."ASiGW-MCC001-bw200-C2: Output"."Dir J2.1.3");
	    
	END_REGION
	
	REGION J2.1.4
	    //J2.1.4
	    #"J2.1.4"(ConveyorID:=_."J2.1.4",
	              ConveyorSensor:=_."ASiGW-MCC001-bw200-C2: Input"."Sensor J2.1.11",
	                   Fault:= DB_UDI.EmptyLine.Fault.Stop.Conveyor[_."J2.1.4"],
	                   Upstream:= DB_UDI.EmptyLine.Upstream.Conveyor[_."J2.1.4"],
	                   Downstream:= DB_UDI.EmptyLine.DownstreamAcu.Stop.Conveyor[_."J2.1.4"],
	                   Interlock:= DB_UDI.EmptyLine.Interlock.Stop.Conveyor[_."J2.1.4"],
	                   RunForward=>_."ASiGW-MCC001-bw200-C2: Output"."Motor J2.1.4",
	                   WriteAsiDir=>_."ASiGW-MCC001-bw200-C2: Output"."Dir J2.1.4");
	
	END_REGION
	
	REGION J2.1.5
	    //J2.1.5
	    #"J2.1.5"(ConveyorID:=_."J2.1.5",
	              ConveyorSensor:=_."ASiGW-MCC001-bw200-C2: Input"."Sensor J2.1.11",
	                   Fault:= DB_UDI.EmptyLine.Fault.Stop.Conveyor[_."J2.1.5"],
	                   Upstream:= DB_UDI.EmptyLine.Upstream.Conveyor[_."J2.1.5"],
	                   Downstream:= DB_UDI.EmptyLine.DownstreamAcu.Stop.Conveyor[_."J2.1.5"],
	                   Interlock:= DB_UDI.EmptyLine.Interlock.Stop.Conveyor[_."J2.1.5"],
	                   RunForward=>_."ASiGW-MCC001-bw200-C2: Output"."Motor J2.1.5",
	                   WriteAsiDir=>_."ASiGW-MCC001-bw200-C2: Output"."Dir J2.1.5");
	
	END_REGION
	
	REGION J2.1.6
	    //J2.1.6
	    #"J2.1.6"(ConveyorID:=_."J2.1.6",
	              ConveyorSensor:=_."ASiGW-MCC001-bw200-C2: Input"."Sensor J2.1.11",
	                   Fault:= DB_UDI.EmptyLine.Fault.Stop.Conveyor[_."J2.1.6"],
	                   Upstream:= DB_UDI.EmptyLine.Upstream.Conveyor[_."J2.1.6"],
	                   Downstream:= DB_UDI.EmptyLine.DownstreamAcu.Stop.Conveyor[_."J2.1.6"],
	                   Interlock:= DB_UDI.EmptyLine.Interlock.Stop.Conveyor[_."J2.1.6"],
	                   RunForward=>_."ASiGW-MCC001-bw200-C2: Output"."Motor J2.1.6",
	                   WriteAsiDir=>_."ASiGW-MCC001-bw200-C2: Output"."Dir J2.1.6");
	
	END_REGION
	
	REGION J2.1.7
	    //J2.1.7
	    #"J2.1.7"(ConveyorID:=_."J2.1.7",
	              ConveyorSensor:=_."ASiGW-MCC001-bw200-C2: Input"."Sensor J2.1.11",
	                   Fault:= DB_UDI.EmptyLine.Fault.Stop.Conveyor[_."J2.1.7"],
	                   Upstream:= DB_UDI.EmptyLine.Upstream.Conveyor[_."J2.1.7"],
	                   Downstream:= DB_UDI.EmptyLine.DownstreamAcu.Stop.Conveyor[_."J2.1.7"],
	                   Interlock:= DB_UDI.EmptyLine.Interlock.Stop.Conveyor[_."J2.1.7"],
	                   RunForward=>_."ASiGW-MCC001-bw200-C2: Output"."Motor J2.1.7",
	                   WriteAsiDir=>_."ASiGW-MCC001-bw200-C2: Output"."Dir J2.1.7");
	
	END_REGION
	
	REGION J2.1.8
	    //J2.1.8
	    #"J2.1.8"(ConveyorID := _."J2.1.8",
	              ConveyorSensor:=_."ASiGW-MCC001-bw200-C2: Input"."Sensor J2.1.11",
	              Fault := DB_UDI.EmptyLine.Fault.Stop.Conveyor[_."J2.1.8"],
	              Upstream := DB_UDI.EmptyLine.Upstream.Conveyor[_."J2.1.8"],
	              Downstream := DB_UDI.EmptyLine.DownstreamAcu.Stop.Conveyor[_."J2.1.8"],
	              Interlock := DB_UDI.EmptyLine.Interlock.Stop.Conveyor[_."J2.1.8"],
	              RunForward => _."ASiGW-MCC001-bw200-C2: Output"."Motor J2.1.8",
	              WriteAsiDir => _."ASiGW-MCC001-bw200-C2: Output"."Dir J2.1.8");
	    
	END_REGION
	
	REGION J2.1.9
	    //J2.1.9
	    #"J2.1.9"(ConveyorID:=_."J2.1.9",
	              ConveyorSensor:=_."ASiGW-MCC001-bw200-C2: Input"."Sensor J2.1.11",
	                   Fault:= DB_UDI.EmptyLine.Fault.Stop.Conveyor[_."J2.1.9"],
	                   Upstream:= DB_UDI.EmptyLine.Upstream.Conveyor[_."J2.1.9"],
	                   Downstream:= DB_UDI.EmptyLine.DownstreamAcu.Stop.Conveyor[_."J2.1.9"],
	                   Interlock:= DB_UDI.EmptyLine.Interlock.Stop.Conveyor[_."J2.1.9"],
	                   RunForward=>_."ASiGW-MCC001-bw200-C2: Output"."Motor J2.1.9",
	                   WriteAsiDir=>_."ASiGW-MCC001-bw200-C2: Output"."Dir J2.1.9");
	
	END_REGION
	
	REGION J2.1.10
	    //J2.1.10
	    #"J2.1.10"(ConveyorID:=_."J2.1.10",
	               ConveyorSensor:=_."ASiGW-MCC001-bw200-C2: Input"."Sensor J2.1.11",
	                   Fault:= DB_UDI.EmptyLine.Fault.Stop.Conveyor[_."J2.1.10"],
	                   Upstream:= DB_UDI.EmptyLine.Upstream.Conveyor[_."J2.1.10"],
	                   Downstream:= DB_UDI.EmptyLine.DownstreamAcu.Stop.Conveyor[_."J2.1.10"],
	                   Interlock:= DB_UDI.EmptyLine.Interlock.Stop.Conveyor[_."J2.1.10"],
	                   RunForward=>_."ASiGW-MCC001-bw200-C2: Output"."Motor J2.1.10",
	                   WriteAsiDir=>_."ASiGW-MCC001-bw200-C2: Output"."Dir J2.1.10");
	
	END_REGION
	
	REGION J2.1.11
	    //J2.1.11
	    #"J2.1.11"(ConveyorID:=_."J2.1.11",
	               ConveyorSensor:=_."ASiGW-MCC001-bw200-C2: Input"."Sensor J2.1.11",
	                   Fault:= DB_UDI.EmptyLine.Fault.Stop.Conveyor[_."J2.1.11"],
	                   Upstream:= DB_UDI.EmptyLine.Upstream.Conveyor[_."J2.1.11"],
	                   Downstream:= DB_UDI.EmptyLine.DownstreamAcu.Stop.Conveyor[_."J2.1.11"],
	                   Interlock:= DB_UDI.EmptyLine.Interlock.Stop.Conveyor[_."J2.1.11"],
	                   RunForward=>_."ASiGW-MCC001-bw200-C2: Output"."Motor J2.1.11",
	                   WriteAsiDir=>_."ASiGW-MCC001-bw200-C2: Output"."Dir J2.1.11");
	
	END_REGION
	
	REGION J2.1.12
	    //J2.1.12
	    #"J2.1.12"(ConveyorID:=_."J2.1.12",
	               ConveyorSensor:=_."ASiGW-MCC001-bw200-C2: Input"."Sensor J2.1.15",
	                   Fault:= DB_UDI.EmptyLine.Fault.Stop.Conveyor[_."J2.1.12"],
	                   Upstream:= DB_UDI.EmptyLine.Upstream.Conveyor[_."J2.1.12"],
	                   Downstream:= DB_UDI.EmptyLine.DownstreamAcu.Stop.Conveyor[_."J2.1.12"],
	                   Interlock:= DB_UDI.EmptyLine.Interlock.Stop.Conveyor[_."J2.1.12"],
	                   RunForward=>_."ASiGW-MCC001-bw200-C2: Output"."Motor J2.1.12",
	                   WriteAsiDir=>_."ASiGW-MCC001-bw200-C2: Output"."Dir J2.1.12");
	
	END_REGION
	
	REGION J2.1.13
	    //J2.1.13
	    #"J2.1.13"(ConveyorID:=_."J2.1.13",
	               ConveyorSensor:=_."ASiGW-MCC001-bw200-C2: Input"."Sensor J2.1.15",
	                   Fault:= DB_UDI.EmptyLine.Fault.Stop.Conveyor[_."J2.1.13"],
	                   Upstream:= DB_UDI.EmptyLine.Upstream.Conveyor[_."J2.1.13"],
	                   Downstream:= DB_UDI.EmptyLine.DownstreamAcu.Stop.Conveyor[_."J2.1.13"],
	                   Interlock:= DB_UDI.EmptyLine.Interlock.Stop.Conveyor[_."J2.1.13"],
	                   RunForward=>_."ASiGW-MCC001-bw200-C2: Output"."Motor J2.1.13",
	                   WriteAsiDir=>_."ASiGW-MCC001-bw200-C2: Output"."Dir J2.1.13");
	
	END_REGION
	
	REGION J2.1.14
	    //J2.1.14
	    #"J2.1.14"(ConveyorID:=_."J2.1.14",
	               ConveyorSensor:=_."ASiGW-MCC001-bw200-C2: Input"."Sensor J2.1.15",
	                   Fault:= DB_UDI.EmptyLine.Fault.Stop.Conveyor[_."J2.1.14"],
	                   Upstream:= DB_UDI.EmptyLine.Upstream.Conveyor[_."J2.1.14"],
	                   Downstream:= DB_UDI.EmptyLine.DownstreamAcu.Stop.Conveyor[_."J2.1.14"],
	                   Interlock:= DB_UDI.EmptyLine.Interlock.Stop.Conveyor[_."J2.1.14"],
	                   RunForward=>_."ASiGW-MCC001-bw200-C2: Output"."Motor J2.1.14",
	                   WriteAsiDir=>_."ASiGW-MCC001-bw200-C2: Output"."Dir J2.1.14");
	        
	END_REGION
	
	REGION J2.1.15
	    //J2.1.15
	    #"J2.1.15"(ConveyorID:=_."J2.1.15",
	               ConveyorSensor:=_."ASiGW-MCC001-bw200-C2: Input"."Sensor J2.1.15",
	                   Fault:= DB_UDI.EmptyLine.Fault.Stop.Conveyor[_."J2.1.15"],
	                   Upstream:= DB_UDI.EmptyLine.Upstream.Conveyor[_."J2.1.15"],
	                   Downstream:= DB_UDI.EmptyLine.DownstreamAcu.Stop.Conveyor[_."J2.1.15"],
	                   Interlock:= DB_UDI.EmptyLine.Interlock.Stop.Conveyor[_."J2.1.15"],
	                   RunForward=>_."ASiGW-MCC001-bw200-C2: Output"."Motor J2.1.15",
	                   WriteAsiDir=>_."ASiGW-MCC001-bw200-C2: Output"."Dir J2.1.15");
	
	END_REGION
	
	REGION J2.2.1
	    //J2.2.1
	    #"J2.2.1"(ConveyorID:=_."J2.2.1",
	                   Fault:= DB_UDI.EmptyLine.Fault.Stop.Conveyor[_."J2.2.1"],
	                   Upstream:= DB_UDI.EmptyLine.Upstream.Conveyor[_."J2.2.1"],
	                   Downstream:= DB_UDI.EmptyLine.DownstreamAcu.Stop.Conveyor[_."J2.2.1"],
	                   Interlock:= DB_UDI.EmptyLine.Interlock.Stop.Conveyor[_."J2.2.1"],
	                   RunForward=>_."ASiGW-MCC001-bw200-C2: Output"."Motor J2.2.1",
	                   WriteAsiDir=>_."ASiGW-MCC001-bw200-C2: Output"."Dir J2.2.1");
	
	END_REGION
	
	REGION J2.2.2
	    //J2.2.2
	    #"J2.2.2"(ConveyorID:=_."J2.2.2",
	              ConveyorSensor:=_."ASiGW-MCC001-bw200-C2: Input"."Sensor J2.2.2",
	                   Fault:= DB_UDI.EmptyLine.Fault.Stop.Conveyor[_."J2.2.2"],
	                   Upstream:= DB_UDI.EmptyLine.Upstream.Conveyor[_."J2.2.2"],
	                   Downstream:= DB_UDI.EmptyLine.DownstreamAcu.Stop.Conveyor[_."J2.2.2"],
	                   Interlock:= DB_UDI.EmptyLine.Interlock.Stop.Conveyor[_."J2.2.2"],
	                   RunForward=>_."ASiGW-MCC001-bw200-C2: Output"."Motor J2.2.2",
	                   WriteAsiDir=>_."ASiGW-MCC001-bw200-C2: Output"."Dir J2.2.2");
	
	END_REGION
	
	REGION J2.3.1
	    //J2.3.1
	    #"J2.3.1"(ConveyorID := _."J2.3.1",
	              ConveyorSensor:=_."ASiGW-MCC001-bw200-C2: Input"."Sensor J2.3.1",
	              Fault := DB_UDI.EmptyLine.Fault.Stop.Conveyor[_."J2.3.1"],
	              Upstream := DB_UDI.EmptyLine.Upstream.Conveyor[_."J2.3.1"],
	              Downstream := DB_UDI.EmptyLine.DownstreamAcu.Stop.Conveyor[_."J2.3.1"],
	              Interlock := DB_UDI.EmptyLine.Interlock.Stop.Conveyor[_."J2.3.1"],
	              RunForward => _."ASiGW-MCC001-bw200-C2: Output"."Motor - J2.3.1",
	              WriteAsiDir => _."ASiGW-MCC001-bw200-C2: Output"."2-25A Dir");
	    
	END_REGION
	
	REGION J2.4.1
	    //J2.4.1 Arm for Merger1
	    #"J2.4.1"(ConveyorID:=_."J2.4.1",
	                   Fault:= DB_UDI.EmptyLine.Fault.Stop.Conveyor[_."J2.4.1"],
	                   Upstream:= DB_UDI.EmptyLine.Upstream.Conveyor[_."J2.4.1"],
	                   Downstream:= DB_UDI.EmptyLine.DownstreamAcu.Stop.Conveyor[_."J2.4.1"],
	                   Interlock:= DB_UDI.EmptyLine.Interlock.Stop.Conveyor[_."J2.4.1"],
	                   RunForward=>_."ASiGW-MCC001-bw200-C2: Output"."Motor J2.4.1",
	                   WriteAsiDir=>_."ASiGW-MCC001-bw200-C2: Output"."Dir J2.4.1");
	
	END_REGION
	
	REGION J1.2.4 Merger
	    //J1.2.4 Merger 1
	    #"J1.2.4"(ConveyorID:=_."J1.2.4",
	              ConveyorSensor:=_."ASiGW-MCC001-bw143-C1: Input"."1-27B I1",
	                   Fault:= DB_UDI.EmptyLine.Fault.Stop.Conveyor[_."J1.2.4"],
	                   Upstream:= DB_UDI.EmptyLine.Upstream.Conveyor[_."J1.2.4"],
	                   Downstream:= DB_UDI.EmptyLine.DownstreamAcu.Stop.Conveyor[_."J1.2.4"],
	                   Interlock:= DB_UDI.EmptyLine.Interlock.Stop.Conveyor[_."J1.2.4"],
	                   RunForward=>_."ASiGW-MCC001-bw143-C1: Output"."Motor J1.2.4",
	                   WriteAsiDir=>_."ASiGW-MCC001-bw143-C1: Output"."Dir J1.2.4");
	         
	END_REGION
	
	REGION J1.2.5
	    //J1.2.5
	    #"J1.2.5"(ConveyorID := _."J1.2.5",
	              ConveyorSensor:=_."ASiGW-MCC001-bw143-C1: Input"."Sensor J1.2.5",
	              Fault := DB_UDI.EmptyLine.Fault.Stop.Conveyor[_."J1.2.5"],
	              Upstream := DB_UDI.EmptyLine.Upstream.Conveyor[_."J1.2.5"],
	              Downstream := DB_UDI.EmptyLine.DownstreamAcu.Stop.Conveyor[_."J1.2.5"],
	              Interlock := DB_UDI.EmptyLine.Interlock.Stop.Conveyor[_."J1.2.5"],
	              RunForward=>_."ASiGW-MCC001-bw143-C1: Output"."Motor J1.2.5",
	              WriteAsiDir=>_."ASiGW-MCC001-bw143-C1: Output"."Dir J1.2.5");
	    
	END_REGION
	
	REGION J1.3.1
	    //J1.3.1
	    #"J1.3.1"(ConveyorID := _."J1.3.1",
	              ConveyorSensor:=_."ASiGW-MCC001-bw143-C1: Input"."Sensor J1.4.7",
	              Fault := DB_UDI.EmptyLine.Fault.Stop.Conveyor[_."J1.3.1"],
	              Upstream := DB_UDI.EmptyLine.Upstream.Conveyor[_."J1.3.1"],
	              Downstream := DB_UDI.EmptyLine.DownstreamAcu.Stop.Conveyor[_."J1.3.1"],
	              Interlock := DB_UDI.EmptyLine.Interlock.Stop.Conveyor[_."J1.3.1"],
	              RunForward=>_."ASiGW-MCC001-bw143-C1: Output"."Motor J1.3.1",
	              WriteAsiDir=>_."ASiGW-MCC001-bw143-C1: Output"."Dir J1.3.1");
	    
	END_REGION
	
	REGION J1.3.2
	    //J1.3.2
	    #"J1.3.2"(ConveyorID:=_."J1.3.2",
	              ConveyorSensor:=_."ASiGW-MCC001-bw143-C1: Input"."Sensor J1.4.7",
	                   Fault:= DB_UDI.EmptyLine.Fault.Stop.Conveyor[_."J1.3.2"],
	                   Upstream:= DB_UDI.EmptyLine.Upstream.Conveyor[_."J1.3.2"],
	                   Downstream:= DB_UDI.EmptyLine.DownstreamAcu.Stop.Conveyor[_."J1.3.2"],
	                   Interlock:= DB_UDI.EmptyLine.Interlock.Stop.Conveyor[_."J1.3.2"],
	                   RunForward=>_."ASiGW-MCC001-bw143-C1: Output"."Motor J1.3.2",
	                   WriteAsiDir=>_."ASiGW-MCC001-bw143-C1: Output"."Dir J1.3.2");
	         
	END_REGION
	
	REGION J1.4.1
	    //J1.4.1
	    #"J1.4.1"(ConveyorID:=_."J1.4.1",
	              ConveyorSensor:=_."ASiGW-MCC001-bw143-C1: Input"."Sensor J1.4.7",
	                   Fault:= DB_UDI.EmptyLine.Fault.Stop.Conveyor[_."J1.4.1"],
	                   Upstream:= DB_UDI.EmptyLine.Upstream.Conveyor[_."J1.4.1"],
	                   Downstream:= DB_UDI.EmptyLine.DownstreamAcu.Stop.Conveyor[_."J1.4.1"],
	                   Interlock:= DB_UDI.EmptyLine.Interlock.Stop.Conveyor[_."J1.4.1"],
	                   RunForward=>_."ASiGW-MCC001-bw143-C1: Output"."Motor J1.4.1",
	                   WriteAsiDir=>_."ASiGW-MCC001-bw143-C1: Output"."Dir J1.4.1");
	         
	END_REGION
	
	REGION J1.4.2
	    //J1.4.2
	    #"J1.4.2"(ConveyorID:=_."J1.4.2",
	              ConveyorSensor:=_."ASiGW-MCC001-bw143-C1: Input"."Sensor J1.4.7",
	                   Fault:= DB_UDI.EmptyLine.Fault.Stop.Conveyor[_."J1.4.2"],
	                   Upstream:= DB_UDI.EmptyLine.Upstream.Conveyor[_."J1.4.2"],
	                   Downstream:= DB_UDI.EmptyLine.DownstreamAcu.Stop.Conveyor[_."J1.4.2"],
	                   Interlock:= DB_UDI.EmptyLine.Interlock.Stop.Conveyor[_."J1.4.2"],
	                   RunForward=>_."ASiGW-MCC001-bw143-C1: Output"."Motor J1.4.2",
	                   WriteAsiDir=>_."ASiGW-MCC001-bw143-C1: Output"."Dir J1.4.2");
	
	END_REGION
	
	REGION J1.4.3
	    //J1.4.3
	    #"J1.4.3"(ConveyorID := _."J1.4.3",
	              ConveyorSensor:=_."ASiGW-MCC001-bw143-C1: Input"."Sensor J1.4.7",
	              Fault := DB_UDI.EmptyLine.Fault.Stop.Conveyor[_."J1.4.3"],
	              Upstream := DB_UDI.EmptyLine.Upstream.Conveyor[_."J1.4.3"],
	              Downstream := DB_UDI.EmptyLine.DownstreamAcu.Stop.Conveyor[_."J1.4.3"],
	              Interlock := DB_UDI.EmptyLine.Interlock.Stop.Conveyor[_."J1.4.3"],
	              RunForward=>_."ASiGW-MCC001-bw143-C1: Output"."Motor J1.4.3",
	              WriteAsiDir=>_."ASiGW-MCC001-bw143-C1: Output"."Dir J1.4.3");
	    
	END_REGION
	
	REGION J1.4.4
	    //J1.4.4
	    #"J1.4.4"(ConveyorID:=_."J1.4.4",
	              ConveyorSensor:=_."ASiGW-MCC001-bw143-C1: Input"."Sensor J1.4.7",
	                   Fault:= DB_UDI.EmptyLine.Fault.Stop.Conveyor[_."J1.4.4"],
	                   Upstream:= DB_UDI.EmptyLine.Upstream.Conveyor[_."J1.4.4"],
	                   Downstream:= DB_UDI.EmptyLine.DownstreamAcu.Stop.Conveyor[_."J1.4.4"],
	                   Interlock:= DB_UDI.EmptyLine.Interlock.Stop.Conveyor[_."J1.4.4"],
	                   RunForward=>_."ASiGW-MCC001-bw143-C1: Output"."Motor J1.4.4",
	                   WriteAsiDir=>_."ASiGW-MCC001-bw143-C1: Output"."Dir J1.4.4");
	
	END_REGION
	
	REGION J1.4.5
	    //J1.4.5
	    #"J1.4.5"(ConveyorID:=_."J1.4.5",
	              ConveyorSensor:=_."ASiGW-MCC001-bw143-C1: Input"."Sensor J1.4.7",
	                   Fault:= DB_UDI.EmptyLine.Fault.Stop.Conveyor[_."J1.4.5"],
	                   Upstream:= DB_UDI.EmptyLine.Upstream.Conveyor[_."J1.4.5"],
	                   Downstream:= DB_UDI.EmptyLine.DownstreamAcu.Stop.Conveyor[_."J1.4.5"],
	                   Interlock:= DB_UDI.EmptyLine.Interlock.Stop.Conveyor[_."J1.4.5"],
	                   RunForward=>_."ASiGW-MCC001-bw143-C1: Output"."Motor J1.4.5",
	                   WriteAsiDir=>_."ASiGW-MCC001-bw143-C1: Output"."Dir J1.4.5");
	END_REGION
	
	REGION J1.4.6
	    //J1.4.6
	    #"J1.4.6"(ConveyorID := _."J1.4.6",
	              ConveyorSensor:=_."ASiGW-MCC001-bw143-C1: Input"."Sensor J1.4.7",
	              Fault := DB_UDI.EmptyLine.Fault.Stop.Conveyor[_."J1.4.6"],
	              Upstream := DB_UDI.EmptyLine.Upstream.Conveyor[_."J1.4.6"],
	              Downstream := DB_UDI.EmptyLine.DownstreamAcu.Stop.Conveyor[_."J1.4.6"],
	              Interlock := DB_UDI.EmptyLine.Interlock.Stop.Conveyor[_."J1.4.6"],
	              RunForward=>_."ASiGW-MCC001-bw143-C1: Output"."Motor J1.4.6",
	              WriteAsiDir=>_."ASiGW-MCC001-bw143-C1: Output"."Dir J1.4.6");
	    
	END_REGION
	
	REGION J1.4.7
	    //J1.4.7
	    #"J1.4.7"(ConveyorID := _."J1.4.7",
	              ConveyorSensor:=_."ASiGW-MCC001-bw143-C1: Input"."Sensor J1.4.7",
	              Fault := DB_UDI.EmptyLine.Fault.Stop.Conveyor[_."J1.4.7"],
	              Upstream := DB_UDI.EmptyLine.Upstream.Conveyor[_."J1.4.7"],
	              Downstream := DB_UDI.EmptyLine.DownstreamAcu.Stop.Conveyor[_."J1.4.7"],
	              Interlock := DB_UDI.EmptyLine.Interlock.Stop.Conveyor[_."J1.4.7"],
	              RunForward => _."ASiGW-MCC001-bw143-C1: Output"."Motor J1.4.7",
	              WriteAsiDir => _."ASiGW-MCC001-bw143-C1: Output"."Dir J1.4.7");
	    
	END_REGION
	
	REGION J1.5.1
	    //J1.5.1
	    #"J1.5.1"(ConveyorID:=_."J1.5.1",
	              ConveyorSensor:=_."ASiGW-MCC001-bw143-C1: Input"."Sensor J1.5.1",
	                   Fault:= DB_UDI.EmptyLine.Fault.Stop.Conveyor[_."J1.5.1"],
	                   Upstream:= DB_UDI.EmptyLine.Upstream.Conveyor[_."J1.5.1"],
	                   Downstream:= DB_UDI.EmptyLine.DownstreamAcu.Stop.Conveyor[_."J1.5.1"],
	                   Interlock:= DB_UDI.EmptyLine.Interlock.Stop.Conveyor[_."J1.5.1"],
	                   RunForward => _."ASiGW-MCC001-bw143-C1: Output"."Motor J1.5.1",
	                   WriteAsiDir => _."ASiGW-MCC001-bw143-C1: Output"."Dir J1.5.1");
	         
	END_REGION
	
	REGION J1.5.2
	    //J1.5.2
	    #"J1.5.2"(ConveyorID := _."J1.5.2",
	              ConveyorSensor:=_."ASiGW-MCC001-bw143-C1: Input"."Sensor J1.5.2",
	              Fault := DB_UDI.EmptyLine.Fault.Stop.Conveyor[_."J1.5.2"],
	              Upstream := DB_UDI.EmptyLine.Upstream.Conveyor[_."J1.5.2"],
	              Downstream := DB_UDI.EmptyLine.DownstreamAcu.Stop.Conveyor[_."J1.5.2"],
	              Interlock := DB_UDI.EmptyLine.Interlock.Stop.Conveyor[_."J1.5.2"],
	              RunForward => _."ASiGW-MCC001-bw143-C1: Output"."Motor J1.5.2",
	              WriteAsiDir => _."ASiGW-MCC001-bw143-C1: Output"."Dir J1.5.2");
	    
	END_REGION
	
	REGION J1.5.3
	    //J1.5.3
	    #"J1.5.3"(ConveyorID:=_."J1.5.3",
	              ConveyorSensor:=_."ASiGW-MCC001-bw143-C1: Input"."Sensor J1.5.3",
	                   Fault:= DB_UDI.EmptyLine.Fault.Stop.Conveyor[_."J1.5.3"],
	                   Upstream:= DB_UDI.EmptyLine.Upstream.Conveyor[_."J1.5.3"],
	                   Downstream:= DB_UDI.EmptyLine.DownstreamAcu.Stop.Conveyor[_."J1.5.3"],
	                   Interlock:= DB_UDI.EmptyLine.Interlock.Stop.Conveyor[_."J1.5.3"],
	                   RunForward => _."ASiGW-MCC001-bw143-C1: Output"."Motor J1.5.3",
	                   WriteAsiDir => _."ASiGW-MCC001-bw143-C1: Output"."Dir J1.5.3");
	
	END_REGION
	
	REGION J1.5.4
	    //J1.5.4
	    #"J1.5.4"(ConveyorID:=_."J1.5.4",
	              ConveyorSensor:=_."ASiGW-MCC001-bw143-C1: Input"."Sensor J1.5.4",
	                   Fault:= DB_UDI.EmptyLine.Fault.Stop.Conveyor[_."J1.5.4"],
	                   Upstream:= DB_UDI.EmptyLine.Upstream.Conveyor[_."J1.5.4"],
	                   Downstream:= DB_UDI.EmptyLine.DownstreamAcu.Stop.Conveyor[_."J1.5.4"],
	                   Interlock:= DB_UDI.EmptyLine.Interlock.Stop.Conveyor[_."J1.5.4"],
	                   RunForward => _."ASiGW-MCC001-bw143-C1: Output"."Motor J1.5.4",
	                   WriteAsiDir => _."ASiGW-MCC001-bw143-C1: Output"."Dir J1.5.4");
	END_REGION
	
	REGION J1.6.1 MABS
	    //Mabs J1.6.1
	    #"J1.6.1"(MABS_ID := _."J1.6.1",
	              ErrorSignal:=DB_UDI."EmptyLine".Fault.Stop.Conveyor[_."J1.6.1"],
	              Upstream:=#"J1.5.4".FilteredSensor,
	              UpstreamRunning := #"J1.5.4".ReadConveyorStatus.Running,
	              Downstream_Straight := #"J1.7.1".FilteredSensor,
	              "Downstream_Right/Left" := #"K1.1.1".FilteredSensor,
	              SortDir := _.EmptyLine.ToteDir.Conveyor[_."J1.6.1"],
	              RemoteOut1:=_."ASiGW-MCC001-bw143-C1: Input"."J1.6.1 -RemoteOut1",
	              RemoteOut2:=_."ASiGW-MCC001-bw143-C1: Input"."J1.6.1 -RemoteOut2",
	              RemoteOut3:=_."ASiGW-MCC001-bw143-C1: Input"."J1.6.1 -RemoteOut3",
	              RemoteOut4:=_."ASiGW-MCC001-bw143-C1: Input"."J1.6.1 -RemoteOut4",
	              Parameter:=DB_ConveyorParameters.Line.EmptyLine.Mabs[_."J1.6.1"],
	              RemoteIn1=>_."ASiGW-MCC001-bw143-C1: Output"."J1.6.1 -RemoteIn1",
	              RemoteIn2=>_."ASiGW-MCC001-bw143-C1: Output"."J1.6.1 -RemoteIn2",
	              RemoteIn3=>_."ASiGW-MCC001-bw143-C1: Output"."J1.6.1 -RemoteIn3",
	              RunWheels=>_."ASiGW-MCC001-bw143-C1: Output"."J1.6.1 -RemoteIn4");
	
	END_REGION
	
	REGION J1.6.2 MABS
	    //Mabs J1.6.2
	    #"J1.6.2"(MABS_ID:=_."J1.6.2",
	              ErrorSignal:=DB_UDI."EmptyLine".Fault.Stop.Conveyor[_."J1.6.2"],
	              Upstream:=#"J1.5.4".FilteredSensor,
	              UpstreamRunning:=#"J1.5.4".ReadConveyorStatus.Running,
	              Downstream_Straight:=#"J1.7.1".FilteredSensor,
	              "Downstream_Right/Left":=#"K1.1.1".FilteredSensor,
	              SortDir:=_.EmptyLine.ToteDir.Conveyor[_."J1.6.2"],
	              RemoteOut1:=_."ASiGW-MCC001-bw143-C1: Input"."J1.6.2 -RemoteOut1",
	              RemoteOut2:=_."ASiGW-MCC001-bw143-C1: Input"."J1.6.2 -RemoteOut2",
	              RemoteOut3:=_."ASiGW-MCC001-bw143-C1: Input"."J1.6.2 -RemoteOut3",
	              RemoteOut4:=_."ASiGW-MCC001-bw143-C1: Input"."J1.6.2 -RemoteOut4",
	              Parameter:=DB_ConveyorParameters.Line.EmptyLine.Mabs[_."J1.6.2"],
	              RemoteIn1=>_."ASiGW-MCC001-bw143-C1: Output"."J1.6.2 -RemoteIn1",
	              RemoteIn2=>_."ASiGW-MCC001-bw143-C1: Output"."J1.6.2 -RemoteIn2",
	              RemoteIn3=>_."ASiGW-MCC001-bw143-C1: Output"."J1.6.2 -RemoteIn3",
	              RunWheels=>_."ASiGW-MCC001-bw143-C1: Output"."J1.6.2 -RemoteIn4");
	
	END_REGION
	
	REGION J1.7.1
	    //J1.7.1 (Go straight )
	    #"J1.7.1"(ConveyorID:=_."J1.7.1",
	              ConveyorSensor:=_."ASiGW-MCC001-bw143-C1: Input"."Sensor J1.7.1",
	                   Fault:= DB_UDI.EmptyLine.Fault.Stop.Conveyor[_."J1.7.1"],
	                   Upstream:= DB_UDI.EmptyLine.Upstream.Conveyor[_."J1.7.1"],
	                   Downstream:= DB_UDI.EmptyLine.DownstreamAcu.Stop.Conveyor[_."J1.7.1"],
	                   Interlock:= DB_UDI.EmptyLine.Interlock.Stop.Conveyor[_."J1.7.1"],
	                   RunForward => _."ASiGW-MCC001-bw143-C1: Output"."Motor J1.7.1",
	                   WriteAsiDir => _."ASiGW-MCC001-bw143-C1: Output"."Dir J1.7.1");
	
	END_REGION
	
	REGION J1.7.2
	    //J1.7.2
	    #"J1.7.2"(ConveyorID := _."J1.7.2",
	              ConveyorSensor:=_."ASiGW-MCC001-bw143-C1: Input"."Sensor J1.7.2",
	              Fault := DB_UDI.EmptyLine.Fault.Stop.Conveyor[_."J1.7.2"],
	              Upstream := DB_UDI.EmptyLine.Upstream.Conveyor[_."J1.7.2"],
	              Downstream := DB_UDI.EmptyLine.DownstreamAcu.Stop.Conveyor[_."J1.7.2"],
	              Interlock := DB_UDI.EmptyLine.Interlock.Stop.Conveyor[_."J1.7.2"],
	              RunForward => _."ASiGW-MCC001-bw143-C1: Output"."Motor J1.7.2",
	              WriteAsiDir => _."ASiGW-MCC001-bw143-C1: Output"."Dir J1.7.2");
	    
	    
	END_REGION
	
	REGION J1.8.1
	    //J1.8.1
	    #"J1.8.1"(ConveyorID:=_."J1.8.1",
	              ConveyorSensor:=_."ASiGW-MCC001-bw143-C1: Input"."Sensor J1.8.1",
	                   Fault:= DB_UDI.EmptyLine.Fault.Stop.Conveyor[_."J1.8.1"],
	                   Upstream:= DB_UDI.EmptyLine.Upstream.Conveyor[_."J1.8.1"],
	                   Downstream:= DB_UDI.EmptyLine.DownstreamAcu.Stop.Conveyor[_."J1.8.1"],
	                   Interlock:= DB_UDI.EmptyLine.Interlock.Stop.Conveyor[_."J1.8.1"],
	                   RunForward => _."ASiGW-MCC001-bw143-C1: Output"."Motor J1.8.1",
	                   WriteAsiDir => _."ASiGW-MCC001-bw143-C1: Output"."Dir J1.8.1");
	         
	END_REGION
	
	REGION J1.8.2
	    //J1.8.2
	    #"J1.8.2"(ConveyorID:=_."J1.8.2",
	              ConveyorSensor:=_."ASiGW-MCC001-bw143-C1: Input"."Sensor J1.8.2",
	                   Fault:= DB_UDI.EmptyLine.Fault.Stop.Conveyor[_."J1.8.2"],
	                   Upstream:= DB_UDI.EmptyLine.Upstream.Conveyor[_."J1.8.2"],
	                   Downstream:= DB_UDI.EmptyLine.DownstreamAcu.Stop.Conveyor[_."J1.8.2"],
	                   Interlock:= DB_UDI.EmptyLine.Interlock.Stop.Conveyor[_."J1.8.2"],
	                   RunForward => _."ASiGW-MCC001-bw143-C1: Output"."Motor J1.8.2",
	                   WriteAsiDir => _."ASiGW-MCC001-bw143-C1: Output"."Dir J1.8.2");
	
	END_REGION
	
	REGION J1.9.1
	    //J1.9.1
	    #"J1.9.1"(ConveyorID:=_."J1.9.1",
	              ConveyorSensor:=_."ASiGW-MCC001-bw143-C1: Input"."Sensor J1.9.1",
	                   Fault:= DB_UDI.EmptyLine.Fault.Stop.Conveyor[_."J1.9.1"],
	                   Upstream:= DB_UDI.EmptyLine.Upstream.Conveyor[_."J1.9.1"],
	                   Downstream:= DB_UDI.EmptyLine.DownstreamAcu.Stop.Conveyor[_."J1.9.1"],
	                   Interlock:= DB_UDI.EmptyLine.Interlock.Stop.Conveyor[_."J1.9.1"],
	                   RunForward => _."ASiGW-MCC001-bw143-C1: Output"."Motor - J1.9.1",
	                   WriteAsiDir => _."ASiGW-MCC001-bw143-C1: Output"."1-5B Dir",
	                   WriteAsiSpeed=>_."ASiGW-MCC001-bw143-C1: Output"."1-5B Speed");
	         
	END_REGION
	
	REGION J1.10.1
	    //J1.10.1
	    #"J1.10.1"(ConveyorID := _."J1.10.1",
	               ConveyorSensor:=_."ASiGW-MCC001-bw143-C1: Input"."Sensor J1.10.1",
	               Fault := DB_UDI.EmptyLine.Fault.Stop.Conveyor[_."J1.10.1"],
	               Upstream := DB_UDI.EmptyLine.Upstream.Conveyor[_."J1.10.1"],
	               Downstream := DB_UDI.EmptyLine.DownstreamAcu.Stop.Conveyor[_."J1.10.1"],
	               Interlock := DB_UDI.EmptyLine.Interlock.Stop.Conveyor[_."J1.10.1"],
	               RunForward => _."ASiGW-MCC001-bw143-C1: Output"."Motor - J1.10.1",
	               WriteAsiDir => _."ASiGW-MCC001-bw143-C1: Output"."1-5B Dir",
	               WriteAsiSpeed => _."ASiGW-MCC001-bw143-C1: Output"."1-5B Speed");
	    
	END_REGION
	
